LIN {X 0,Y 480.607,Z 857.054,A -85,B 0,C 180,E1 -14352.742,E2 -14352.742} C_VEL
LIN {X 0,Y 484.902,Z 835.629,A -85,B 0,C 180,E1 -14353.946,E2 -14353.946} C_VEL
LIN {X 0,Y 488.749,Z 813.876,A -85,B 0,C 180,E1 -14354.976,E2 -14354.976} C_VEL
LIN {X 0,Y 492.238,Z 790.021,A -85,B 0,C 180,E1 -14355.873,E2 -14355.873} C_VEL
LIN {X 0,Y 494.835,Z 768.166,A -85,B 0,C 180,E1 -14356.519,E2 -14356.519} C_VEL
LIN {X 0,Y 497.066,Z 742.106,A -85,B 0,C 180,E1 -14357.081,E2 -14357.081} C_VEL
LIN {X 0,Y 507.784,Z 512.286,A -85,B 0,C 180,E1 -14360.624,E2 -14360.624} C_VEL
LIN {X 0,Y 509.838,Z 466.585,A -85,B 0,C 180,E1 -14361.344,E2 -14361.344} C_VEL
LIN {X 0,Y 502.67,Z 455.07,A -85,B 0,C 180,E1 -14362.649,E2 -14362.649} C_VEL
LIN {X 0,Y 491.609,Z 438.773,A -85,B 0,C 180,E1 -14364.787,E2 -14364.787} C_VEL
LIN {X 0,Y 480.959,Z 424.124,A -85,B 0,C 180,E1 -14367.032,E2 -14367.032} C_VEL
LIN {X 0,Y 472.701,Z 413.452,A -85,B 0,C 180,E1 -14368.927,E2 -14368.927} C_VEL
LIN {X 0,Y 468.353,Z 407.951,A -85,B 0,C 180,E1 -14369.993,E2 -14369.993} C_VEL
LIN {X 0,Y 464.571,Z 403.2,A -85,B 0,C 180,E1 -14370.965,E2 -14370.965} C_VEL
LIN {X 0,Y 460.387,Z 398.04,A -85,B 0,C 180,E1 -14372.093,E2 -14372.093} C_VEL
LIN {X 0,Y 456.745,Z 393.676,A -85,B 0,C 180,E1 -14373.124,E2 -14373.124} C_VEL
LIN {X 0,Y 455.561,Z 392.247,A -85,B 0,C 180,E1 -14373.471,E2 -14373.471} C_VEL
LIN {X 0,Y 452.156,Z 388.527,A -85,B 0,C 180,E1 -14374.49,E2 -14374.49} C_VEL
LIN {X 0,Y 450.792,Z 386.471,A -85,B 0,C 180,E1 -14374.934,E2 -14374.934} C_VEL
LIN {X 0,Y 447.515,Z 383.478,A -85,B 0,C 180,E1 -14375.971,E2 -14375.971} C_VEL
LIN {X 0,Y 445.396,Z 380.169,A -85,B 0,C 180,E1 -14376.727,E2 -14376.727} C_VEL
LIN {X 0,Y 442.222,Z 377.701,A -85,B 0,C 180,E1 -14377.815,E2 -14377.815} C_VEL
LIN {X 0,Y 440.297,Z 374.242,A -85,B 0,C 180,E1 -14378.595,E2 -14378.595} C_VEL
LIN {X 0,Y 439.743,Z 373.706,A -85,B 0,C 180,E1 -14378.805,E2 -14378.805} C_VEL
LIN {X 0,Y 436.653,Z 371.721,A -85,B 0,C 180,E1 -14379.98,E2 -14379.98} C_VEL
LIN {X 0,Y 434.814,Z 368.919,A -85,B 0,C 180,E1 -14380.801,E2 -14380.801} C_VEL
LIN {X 0,Y 434.363,Z 367.099,A -85,B 0,C 180,E1 -14381.105,E2 -14381.105} C_VEL
LIN {X 0,Y 434.359,Z 367.094,A -85,B 0,C 180,E1 -14384.922,E2 -14384.922} C_VEL
LIN {X 0,Y 434.379,Z 367.091,A -85,B 0,C 180,E1 -14388.582,E2 -14388.582} C_VEL
LIN {X 0,Y 434.41,Z 367.102,A -85,B 0,C 180,E1 -14392.328,E2 -14392.328} C_VEL
LIN {X 0,Y 434.406,Z 367.121,A -85,B 0,C 180,E1 -14396.173,E2 -14396.173} C_VEL
LIN {X 0,Y 434.379,Z 367.105,A -85,B 0,C 180,E1 -14399.868,E2 -14399.868} C_VEL
LIN {X 0,Y 434.36,Z 367.091,A -85,B 0,C 180,E1 -14403.563,E2 -14403.563} C_VEL
LIN {X 0,Y 434.358,Z 367.094,A -85,B 0,C 180,E1 -14407.274,E2 -14407.274} C_VEL
LIN {X 0,Y 434.385,Z 367.106,A -85,B 0,C 180,E1 -14410.88,E2 -14410.88} C_VEL
LIN {X 0,Y 434.417,Z 367.117,A -85,B 0,C 180,E1 -14414.666,E2 -14414.666} C_VEL
LIN {X 0,Y 434.406,Z 367.116,A -85,B 0,C 180,E1 -14418.52,E2 -14418.52} C_VEL
LIN {X 0,Y 434.457,Z 367.443,A -85,B 0,C 180,E1 -14418.657,E2 -14418.657} C_VEL
LIN {X 0,Y 435.442,Z 370.22,A -85,B 0,C 180,E1 -14419.17,E2 -14419.17} C_VEL
LIN {X 0,Y 437.864,Z 372.753,A -85,B 0,C 180,E1 -14420.171,E2 -14420.171} C_VEL
LIN {X 0,Y 440.192,Z 374.091,A -85,B 0,C 180,E1 -14421.032,E2 -14421.032} C_VEL
LIN {X 0,Y 442.012,Z 377.461,A -85,B 0,C 180,E1 -14421.777,E2 -14421.777} C_VEL
LIN {X 0,Y 445.345,Z 380.151,A -85,B 0,C 180,E1 -14422.926,E2 -14422.926} C_VEL
LIN {X 0,Y 448.828,Z 384.901,A -85,B 0,C 180,E1 -14424.129,E2 -14424.129} C_VEL
LIN {X 0,Y 450.868,Z 387.155,A -85,B 0,C 180,E1 -14424.781,E2 -14424.781} C_VEL
LIN {X 0,Y 454.843,Z 392.158,A -85,B 0,C 180,E1 -14426.012,E2 -14426.012} C_VEL
LIN {X 0,Y 459.096,Z 397.573,A -85,B 0,C 180,E1 -14427.253,E2 -14427.253} C_VEL
LIN {X 0,Y 466.167,Z 406.901,A -85,B 0,C 180,E1 -14429.172,E2 -14429.172} C_VEL
LIN {X 0,Y 473.965,Z 417.836,A -85,B 0,C 180,E1 -14431.122,E2 -14431.122} C_VEL
LIN {X 0,Y 482.316,Z 429.887,A -85,B 0,C 180,E1 -14433.04,E2 -14433.04} C_VEL
LIN {X 0,Y 491.291,Z 443.78,A -85,B 0,C 180,E1 -14434.954,E2 -14434.954} C_VEL
LIN {X 0,Y 501.111,Z 459.807,A -85,B 0,C 180,E1 -14436.895,E2 -14436.895} C_VEL
LIN {X 0,Y 509.771,Z 475.225,A -85,B 0,C 180,E1 -14438.507,E2 -14438.507} C_VEL
LIN {X 0,Y 498.368,Z 722.255,A -85,B 0,C 180,E1 -14442.296,E2 -14442.296} C_VEL
LIN {X 0,Y 496.144,Z 766.257,A -85,B 0,C 180,E1 -14443.004,E2 -14443.004} C_VEL
LIN {X 0,Y 493.733,Z 790.305,A -85,B 0,C 180,E1 -14443.551,E2 -14443.551} C_VEL
LIN {X 0,Y 490.946,Z 811.995,A -85,B 0,C 180,E1 -14444.195,E2 -14444.195} C_VEL
LIN {X 0,Y 487.211,Z 835.448,A -85,B 0,C 180,E1 -14445.091,E2 -14445.091} C_VEL
LIN {X 0,Y 483.594,Z 855.156,A -85,B 0,C 180,E1 -14446.016,E2 -14446.016} C_VEL
LIN {X 0,Y 478.87,Z 878.071,A -85,B 0,C 180,E1 -14447.306,E2 -14447.306} C_VEL
LIN {X 0,Y 474.326,Z 897.652,A -85,B 0,C 180,E1 -14448.63,E2 -14448.63} C_VEL
LIN {X 0,Y 469.589,Z 916.875,A -85,B 0,C 180,E1 -14450.14,E2 -14450.14} C_VEL
LIN {X 0,Y 464.072,Z 937.548,A -85,B 0,C 180,E1 -14452.054,E2 -14452.054} C_VEL
LIN {X 0,Y 459.269,Z 954.903,A -85,B 0,C 180,E1 -14453.92,E2 -14453.92} C_VEL
LIN {X 0,Y 453.924,Z 973.715,A -85,B 0,C 180,E1 -14456.282,E2 -14456.282} C_VEL
LIN {X 0,Y 449.837,Z 988.033,A -85,B 0,C 180,E1 -14458.36,E2 -14458.36} C_VEL
LIN {X 0,Y 445.405,Z 1003.835,A -85,B 0,C 180,E1 -14460.994,E2 -14460.994} C_VEL
LIN {X 0,Y 441.88,Z 1016.82,A -85,B 0,C 180,E1 -14463.527,E2 -14463.527} C_VEL
LIN {X 0,Y 438.683,Z 1029.589,A -85,B 0,C 180,E1 -14466.389,E2 -14466.389} C_VEL
LIN {X 0,Y 436.18,Z 1040.548,A -85,B 0,C 180,E1 -14469.327,E2 -14469.327} C_VEL
LIN {X 0,Y 434.432,Z 1049.638,A -85,B 0,C 180,E1 -14472.175,E2 -14472.175} C_VEL
LIN {X 0,Y 433.099,Z 1058.109,A -85,B 0,C 180,E1 -14475.425,E2 -14475.425} C_VEL
LIN {X 0,Y 432.416,Z 1064.059,A -85,B 0,C 180,E1 -14478.259,E2 -14478.259} C_VEL
LIN {X 0,Y 432.041,Z 1069.434,A -85,B 0,C 180,E1 -14481.616,E2 -14481.616} C_VEL
LIN {X 0,Y 431.949,Z 1072.492,A -85,B 0,C 180,E1 -14484.421,E2 -14484.421} C_VEL
LIN {X 0,Y 431.945,Z 1074.289,A -85,B 0,C 180,E1 -14487.081,E2 -14487.081} C_VEL
LIN {X 0,Y 431.946,Z 1074.998,A -85,B 0,C 180,E1 -14490.265,E2 -14490.265} C_VEL
LIN {X 0,Y 431.947,Z 1074.217,A -85,B 0,C 180,E1 -14493.052,E2 -14493.052} C_VEL
LIN {X 0,Y 431.952,Z 1072.37,A -85,B 0,C 180,E1 -14495.712,E2 -14495.712} C_VEL
LIN {X 0,Y 432.06,Z 1068.893,A -85,B 0,C 180,E1 -14498.816,E2 -14498.816} C_VEL
LIN {X 0,Y 432.44,Z 1063.789,A -85,B 0,C 180,E1 -14501.875,E2 -14501.875} C_VEL
LIN {X 0,Y 433.14,Z 1057.785,A -85,B 0,C 180,E1 -14504.71,E2 -14504.71} C_VEL
LIN {X 0,Y 434.569,Z 1048.793,A -85,B 0,C 180,E1 -14508.096,E2 -14508.096} C_VEL
LIN {X 0,Y 436.279,Z 1040.061,A -85,B 0,C 180,E1 -14510.808,E2 -14510.808} C_VEL
LIN {X 0,Y 438.984,Z 1028.25,A -85,B 0,C 180,E1 -14513.918,E2 -14513.918} C_VEL
LIN {X 0,Y 442.043,Z 1016.141,A -85,B 0,C 180,E1 -14516.607,E2 -14516.607} C_VEL
LIN {X 0,Y 446.02,Z 1001.585,A -85,B 0,C 180,E1 -14519.403,E2 -14519.403} C_VEL
LIN {X 0,Y 450.069,Z 987.118,A -85,B 0,C 180,E1 -14521.771,E2 -14521.771} C_VEL
LIN {X 0,Y 454.46,Z 971.776,A -85,B 0,C 180,E1 -14523.976,E2 -14523.976} C_VEL
LIN {X 0,Y 459.719,Z 953.135,A -85,B 0,C 180,E1 -14526.271,E2 -14526.271} C_VEL
LIN {X 0,Y 464.436,Z 936.092,A -85,B 0,C 180,E1 -14528.083,E2 -14528.083} C_VEL
LIN {X 0,Y 470.052,Z 914.786,A -85,B 0,C 180,E1 -14530.022,E2 -14530.022} C_VEL
LIN {X 0,Y 474.493,Z 896.72,A -85,B 0,C 180,E1 -14531.428,E2 -14531.428} C_VEL
LIN {X 0,Y 479.379,Z 875.572,A -85,B 0,C 180,E1 -14532.841,E2 -14532.841} C_VEL
LIN {X 0,Y 483.777,Z 853.85,A -85,B 0,C 180,E1 -14534.042,E2 -14534.042} C_VEL
LIN {X 0,Y 487.42,Z 833.905,A -85,B 0,C 180,E1 -14534.967,E2 -14534.967} C_VEL
LIN {X 0,Y 491.276,Z 808.969,A -85,B 0,C 180,E1 -14535.894,E2 -14535.894} C_VEL
LIN {X 0,Y 493.87,Z 788.534,A -85,B 0,C 180,E1 -14536.486,E2 -14536.486} C_VEL
LIN {X 0,Y 496.258,Z 763.311,A -85,B 0,C 180,E1 -14537.04,E2 -14537.04} C_VEL
LIN {X 0,Y 499.532,Z 694.355,A -85,B 0,C 180,E1 -14538.123,E2 -14538.123} C_VEL
LIN {X 0,Y 509.617,Z 474.877,A -85,B 0,C 180,E1 -14541.5,E2 -14541.5} C_VEL
LIN {X 0,Y 498.824,Z 456.036,A -85,B 0,C 180,E1 -14543.517,E2 -14543.517} C_VEL
LIN {X 0,Y 487.736,Z 438.217,A -85,B 0,C 180,E1 -14545.754,E2 -14545.754} C_VEL
LIN {X 0,Y 476.706,Z 421.573,A -85,B 0,C 180,E1 -14548.197,E2 -14548.197} C_VEL
LIN {X 0,Y 467.195,Z 408.431,A -85,B 0,C 180,E1 -14550.512,E2 -14550.512} C_VEL
LIN {X 0,Y 461.589,Z 400.928,A -85,B 0,C 180,E1 -14551.997,E2 -14551.997} C_VEL
LIN {X 0,Y 457.333,Z 395.328,A -85,B 0,C 180,E1 -14553.196,E2 -14553.196} C_VEL
LIN {X 0,Y 452.168,Z 388.749,A -85,B 0,C 180,E1 -14554.746,E2 -14554.746} C_VEL
LIN {X 0,Y 449.208,Z 385.26,A -85,B 0,C 180,E1 -14555.682,E2 -14555.682} C_VEL
LIN {X 0,Y 446.351,Z 381.674,A -85,B 0,C 180,E1 -14556.64,E2 -14556.64} C_VEL
LIN {X 0,Y 445.112,Z 380.025,A -85,B 0,C 180,E1 -14557.074,E2 -14557.074} C_VEL
LIN {X 0,Y 441.822,Z 377.223,A -85,B 0,C 180,E1 -14558.213,E2 -14558.213} C_VEL
LIN {X 0,Y 440.006,Z 373.768,A -85,B 0,C 180,E1 -14558.958,E2 -14558.958} C_VEL
LIN {X 0,Y 436.552,Z 371.673,A -85,B 0,C 180,E1 -14560.255,E2 -14560.255} C_VEL
LIN {X 0,Y 434.855,Z 368.973,A -85,B 0,C 180,E1 -14561.012,E2 -14561.012} C_VEL
LIN {X 0,Y 434.41,Z 367.108,A -85,B 0,C 180,E1 -14561.306,E2 -14561.306} C_VEL
LIN {X 0,Y 434.389,Z 367.101,A -85,B 0,C 180,E1 -14565.06,E2 -14565.06} C_VEL
LIN {X 0,Y 434.365,Z 367.094,A -85,B 0,C 180,E1 -14568.716,E2 -14568.716} C_VEL
LIN {X 0,Y 434.361,Z 367.092,A -85,B 0,C 180,E1 -14572.46,E2 -14572.46} C_VEL
LIN {X 0,Y 434.378,Z 367.102,A -85,B 0,C 180,E1 -14576.172,E2 -14576.172} C_VEL
LIN {X 0,Y 434.412,Z 367.12,A -85,B 0,C 180,E1 -14579.868,E2 -14579.868} C_VEL
LIN {X 0,Y 434.407,Z 367.106,A -85,B 0,C 180,E1 -14583.695,E2 -14583.695} C_VEL
LIN {X 0,Y 434.387,Z 367.09,A -85,B 0,C 180,E1 -14587.406,E2 -14587.406} C_VEL
LIN {X 0,Y 434.365,Z 367.093,A -85,B 0,C 180,E1 -14591.015,E2 -14591.015} C_VEL
LIN {X 0,Y 434.368,Z 367.102,A -85,B 0,C 180,E1 -14594.804,E2 -14594.804} C_VEL
LIN {X 0,Y 434.386,Z 367.113,A -85,B 0,C 180,E1 -14598.521,E2 -14598.521} C_VEL
LIN {X 0,Y 434.391,Z 367.263,A -85,B 0,C 180,E1 -14599.146,E2 -14599.146} C_VEL
LIN {X 0,Y 435.315,Z 369.953,A -85,B 0,C 180,E1 -14599.629,E2 -14599.629} C_VEL
LIN {X 0,Y 437.809,Z 372.717,A -85,B 0,C 180,E1 -14600.662,E2 -14600.662} C_VEL
LIN {X 0,Y 440.238,Z 374.085,A -85,B 0,C 180,E1 -14601.554,E2 -14601.554} C_VEL
LIN {X 0,Y 442.066,Z 377.526,A -85,B 0,C 180,E1 -14602.298,E2 -14602.298} C_VEL
LIN {X 0,Y 444.961,Z 379.949,A -85,B 0,C 180,E1 -14603.297,E2 -14603.297} C_VEL
LIN {X 0,Y 445.862,Z 380.7,A -85,B 0,C 180,E1 -14603.597,E2 -14603.597} C_VEL
LIN {X 0,Y 448.273,Z 384.397,A -85,B 0,C 180,E1 -14604.442,E2 -14604.442} C_VEL
LIN {X 0,Y 451.31,Z 387.146,A -85,B 0,C 180,E1 -14605.386,E2 -14605.386} C_VEL
LIN {X 0,Y 454.326,Z 391.184,A -85,B 0,C 180,E1 -14606.325,E2 -14606.325} C_VEL
LIN {X 0,Y 456.534,Z 393.368,A -85,B 0,C 180,E1 -14606.96,E2 -14606.96} C_VEL
LIN {X 0,Y 459.957,Z 397.656,A -85,B 0,C 180,E1 -14607.935,E2 -14607.935} C_VEL
LIN {X 0,Y 461.627,Z 399.54,A -85,B 0,C 180,E1 -14608.388,E2 -14608.388} C_VEL
LIN {X 0,Y 466.733,Z 405.915,A -85,B 0,C 180,E1 -14609.732,E2 -14609.732} C_VEL
LIN {X 0,Y 471.262,Z 411.659,A -85,B 0,C 180,E1 -14610.859,E2 -14610.859} C_VEL
LIN {X 0,Y 478.641,Z 421.069,A -85,B 0,C 180,E1 -14612.578,E2 -14612.578} C_VEL
LIN {X 0,Y 489.178,Z 435.437,A -85,B 0,C 180,E1 -14614.841,E2 -14614.841} C_VEL
LIN {X 0,Y 500.544,Z 451.857,A -85,B 0,C 180,E1 -14617.069,E2 -14617.069} C_VEL
LIN {X 0,Y 509.147,Z 465.502,A -85,B 0,C 180,E1 -14618.646,E2 -14618.646} C_VEL
LIN {X 0,Y 509.876,Z 467.057,A -85,B 0,C 180,E1 -14618.784,E2 -14618.784} C_VEL
LIN {X 0,Y 498.05,Z 722.14,A -85,B 0,C 180,E1 -14622.693,E2 -14622.693} C_VEL
LIN {X 0,Y 496.16,Z 753.273,A -85,B 0,C 180,E1 -14623.235,E2 -14623.235} C_VEL
LIN {X 0,Y 494.016,Z 774.953,A -85,B 0,C 180,E1 -14623.763,E2 -14623.763} C_VEL
LIN {X 0,Y 490.73,Z 800.447,A -85,B 0,C 180,E1 -14624.592,E2 -14624.592} C_VEL
LIN {X 0,Y 487.43,Z 821.156,A -85,B 0,C 180,E1 -14625.448,E2 -14625.448} C_VEL
LIN {X 0,Y 483.211,Z 844.209,A -85,B 0,C 180,E1 -14626.607,E2 -14626.607} C_VEL
LIN {X 0,Y 478.889,Z 864.397,A -85,B 0,C 180,E1 -14627.836,E2 -14627.836} C_VEL
LIN {X 0,Y 474.078,Z 885.286,A -85,B 0,C 180,E1 -14629.329,E2 -14629.329} C_VEL
LIN {X 0,Y 468.947,Z 905.227,A -85,B 0,C 180,E1 -14631.024,E2 -14631.024} C_VEL
LIN {X 0,Y 464.194,Z 922.816,A -85,B 0,C 180,E1 -14632.751,E2 -14632.751} C_VEL
LIN {X 0,Y 458.768,Z 941.82,A -85,B 0,C 180,E1 -14634.93,E2 -14634.93} C_VEL
LIN {X 0,Y 454.185,Z 957.46,A -85,B 0,C 180,E1 -14637.011,E2 -14637.011} C_VEL
LIN {X 0,Y 449.179,Z 974.473,A -85,B 0,C 180,E1 -14639.648,E2 -14639.648} C_VEL
LIN {X 0,Y 445.35,Z 987.585,A -85,B 0,C 180,E1 -14642.015,E2 -14642.015} C_VEL
LIN {X 0,Y 441.421,Z 1001.642,A -85,B 0,C 180,E1 -14644.968,E2 -14644.968} C_VEL
LIN {X 0,Y 438.583,Z 1012.347,A -85,B 0,C 180,E1 -14647.621,E2 -14647.621} C_VEL
LIN {X 0,Y 436.08,Z 1023.008,A -85,B 0,C 180,E1 -14650.721,E2 -14650.721} C_VEL
LIN {X 0,Y 434.355,Z 1031.358,A -85,B 0,C 180,E1 -14653.689,E2 -14653.689} C_VEL
LIN {X 0,Y 433.163,Z 1038.583,A -85,B 0,C 180,E1 -14656.79,E2 -14656.79} C_VEL
LIN {X 0,Y 432.436,Z 1044.258,A -85,B 0,C 180,E1 -14660.014,E2 -14660.014} C_VEL
LIN {X 0,Y 432.129,Z 1047.959,A -85,B 0,C 180,E1 -14662.822,E2 -14662.822} C_VEL
LIN {X 0,Y 432.054,Z 1049.16,A -85,B 0,C 180,E1 -14664.016,E2 -14664.016} C_VEL
LIN {X 0,Y 431.001,Z 1050.055,A -85,B 0,C 180,E1 -14665.031,E2 -14665.031} C_VEL
LIN {X 0,Y 426.312,Z 1051.369,A -85,B 0,C 180,E1 -14666.947,E2 -14666.947} C_VEL
LIN {X 0,Y 424.146,Z 1051.897,A -85,B 0,C 180,E1 -14668.194,E2 -14668.194} C_VEL
LIN {X 0,Y 423.955,Z 1051.968,A -85,B 0,C 180,E1 -14668.646,E2 -14668.646} C_VEL
LIN {X 0,Y 423.958,Z 1051.984,A -85,B 0,C 180,E1 -14671.352,E2 -14671.352} C_VEL
LIN {X 0,Y 424.005,Z 1050.767,A -85,B 0,C 180,E1 -14674.463,E2 -14674.463} C_VEL
LIN {X 0,Y 424.156,Z 1047.974,A -85,B 0,C 180,E1 -14677.586,E2 -14677.586} C_VEL
LIN {X 0,Y 424.506,Z 1044.214,A -85,B 0,C 180,E1 -14680.45,E2 -14680.45} C_VEL
LIN {X 0,Y 425.318,Z 1038.416,A -85,B 0,C 180,E1 -14683.736,E2 -14683.736} C_VEL
LIN {X 0,Y 426.557,Z 1031.476,A -85,B 0,C 180,E1 -14686.758,E2 -14686.758} C_VEL
LIN {X 0,Y 428.508,Z 1022.705,A -85,B 0,C 180,E1 -14689.918,E2 -14689.918} C_VEL
LIN {X 0,Y 431.068,Z 1012.367,A -85,B 0,C 180,E1 -14692.946,E2 -14692.946} C_VEL
LIN {X 0,Y 434.273,Z 1000.957,A -85,B 0,C 180,E1 -14695.808,E2 -14695.808} C_VEL
LIN {X 0,Y 438.198,Z 987.585,A -85,B 0,C 180,E1 -14698.632,E2 -14698.632} C_VEL
LIN {X 0,Y 442.219,Z 974.448,A -85,B 0,C 180,E1 -14701.033,E2 -14701.033} C_VEL
LIN {X 0,Y 447.368,Z 957.672,A -85,B 0,C 180,E1 -14703.662,E2 -14703.662} C_VEL
LIN {X 0,Y 452.053,Z 942.317,A -85,B 0,C 180,E1 -14705.731,E2 -14705.731} C_VEL
LIN {X 0,Y 457.887,Z 922.629,A -85,B 0,C 180,E1 -14708.011,E2 -14708.011} C_VEL
LIN {X 0,Y 462.685,Z 905.512,A -85,B 0,C 180,E1 -14709.705,E2 -14709.705} C_VEL
LIN {X 0,Y 468.004,Z 885.543,A -85,B 0,C 180,E1 -14711.417,E2 -14711.417} C_VEL
LIN {X 0,Y 472.925,Z 864.871,A -85,B 0,C 180,E1 -14712.906,E2 -14712.906} C_VEL
LIN {X 0,Y 477.606,Z 843.711,A -85,B 0,C 180,E1 -14714.199,E2 -14714.199} C_VEL
LIN {X 0,Y 481.741,Z 821.735,A -85,B 0,C 180,E1 -14715.307,E2 -14715.307} C_VEL
LIN {X 0,Y 485.173,Z 800.872,A -85,B 0,C 180,E1 -14716.175,E2 -14716.175} C_VEL
LIN {X 0,Y 488.609,Z 774.994,A -85,B 0,C 180,E1 -14717.02,E2 -14717.02} C_VEL
LIN {X 0,Y 490.823,Z 753.157,A -85,B 0,C 180,E1 -14717.553,E2 -14717.553} C_VEL
LIN {X 0,Y 492.819,Z 720.765,A -85,B 0,C 180,E1 -14718.115,E2 -14718.115} C_VEL
LIN {X 0,Y 504.833,Z 470.537,A -85,B 0,C 180,E1 -14721.974,E2 -14721.974} C_VEL
LIN {X 0,Y 494.554,Z 454.342,A -85,B 0,C 180,E1 -14723.924,E2 -14723.924} C_VEL
LIN {X 0,Y 483.467,Z 438.399,A -85,B 0,C 180,E1 -14726.197,E2 -14726.197} C_VEL
LIN {X 0,Y 473.671,Z 425.178,A -85,B 0,C 180,E1 -14728.396,E2 -14728.396} C_VEL
LIN {X 0,Y 465.75,Z 414.967,A -85,B 0,C 180,E1 -14730.34,E2 -14730.34} C_VEL
LIN {X 0,Y 461.801,Z 410.002,A -85,B 0,C 180,E1 -14731.376,E2 -14731.376} C_VEL
LIN {X 0,Y 457.778,Z 405.021,A -85,B 0,C 180,E1 -14732.486,E2 -14732.486} C_VEL
LIN {X 0,Y 454.017,Z 400.251,A -85,B 0,C 180,E1 -14733.585,E2 -14733.585} C_VEL
LIN {X 0,Y 449.874,Z 395.681,A -85,B 0,C 180,E1 -14734.845,E2 -14734.845} C_VEL
LIN {X 0,Y 448.515,Z 393.78,A -85,B 0,C 180,E1 -14735.291,E2 -14735.291} C_VEL
LIN {X 0,Y 445.049,Z 390.259,A -85,B 0,C 180,E1 -14736.427,E2 -14736.427} C_VEL
LIN {X 0,Y 443.377,Z 387.689,A -85,B 0,C 180,E1 -14737.036,E2 -14737.036} C_VEL
LIN {X 0,Y 440.106,Z 384.859,A -85,B 0,C 180,E1 -14738.194,E2 -14738.194} C_VEL
LIN {X 0,Y 438.141,Z 381.457,A -85,B 0,C 180,E1 -14739.004,E2 -14739.004} C_VEL
LIN {X 0,Y 434.79,Z 379.107,A -85,B 0,C 180,E1 -14740.311,E2 -14740.311} C_VEL
LIN {X 0,Y 432.787,Z 375.962,A -85,B 0,C 180,E1 -14741.233,E2 -14741.233} C_VEL
LIN {X 0,Y 432.209,Z 374.803,A -85,B 0,C 180,E1 -14741.522,E2 -14741.522} C_VEL
LIN {X 0,Y 428.816,Z 372.879,A -85,B 0,C 180,E1 -14743.054,E2 -14743.054} C_VEL
LIN {X 0,Y 426.978,Z 370.049,A -85,B 0,C 180,E1 -14744.063,E2 -14744.063} C_VEL
LIN {X 0,Y 426.441,Z 368.079,A -85,B 0,C 180,E1 -14744.496,E2 -14744.496} C_VEL
LIN {X 0,Y 426.465,Z 368.081,A -85,B 0,C 180,E1 -14748.23,E2 -14748.23} C_VEL
LIN {X 0,Y 426.481,Z 368.092,A -85,B 0,C 180,E1 -14752.185,E2 -14752.185} C_VEL
LIN {X 0,Y 426.464,Z 368.111,A -85,B 0,C 180,E1 -14756.101,E2 -14756.101} C_VEL
LIN {X 0,Y 426.44,Z 368.092,A -85,B 0,C 180,E1 -14759.866,E2 -14759.866} C_VEL
LIN {X 0,Y 426.423,Z 368.08,A -85,B 0,C 180,E1 -14763.63,E2 -14763.63} C_VEL
LIN {X 0,Y 426.418,Z 368.081,A -85,B 0,C 180,E1 -14767.41,E2 -14767.41} C_VEL
LIN {X 0,Y 426.426,Z 368.09,A -85,B 0,C 180,E1 -14771.223,E2 -14771.223} C_VEL
LIN {X 0,Y 426.447,Z 368.1,A -85,B 0,C 180,E1 -14774.979,E2 -14774.979} C_VEL
LIN {X 0,Y 426.456,Z 368.293,A -85,B 0,C 180,E1 -14775.247,E2 -14775.247} C_VEL
LIN {X 0,Y 427.321,Z 370.893,A -85,B 0,C 180,E1 -14775.819,E2 -14775.819} C_VEL
LIN {X 0,Y 429.991,Z 373.788,A -85,B 0,C 180,E1 -14777.177,E2 -14777.177} C_VEL
LIN {X 0,Y 432.52,Z 375.161,A -85,B 0,C 180,E1 -14778.29,E2 -14778.29} C_VEL
LIN {X 0,Y 434.16,Z 378.422,A -85,B 0,C 180,E1 -14779.089,E2 -14779.089} C_VEL
LIN {X 0,Y 436.932,Z 380.842,A -85,B 0,C 180,E1 -14780.216,E2 -14780.216} C_VEL
LIN {X 0,Y 438.24,Z 381.718,A -85,B 0,C 180,E1 -14780.711,E2 -14780.711} C_VEL
LIN {X 0,Y 440.548,Z 385.401,A -85,B 0,C 180,E1 -14781.643,E2 -14781.643} C_VEL
LIN {X 0,Y 443.841,Z 388.254,A -85,B 0,C 180,E1 -14782.798,E2 -14782.798} C_VEL
LIN {X 0,Y 446.775,Z 392.266,A -85,B 0,C 180,E1 -14783.826,E2 -14783.826} C_VEL
LIN {X 0,Y 449.151,Z 395.008,A -85,B 0,C 180,E1 -14784.601,E2 -14784.601} C_VEL
LIN {X 0,Y 452.706,Z 399.589,A -85,B 0,C 180,E1 -14785.722,E2 -14785.722} C_VEL
LIN {X 0,Y 456.806,Z 404.898,A -85,B 0,C 180,E1 -14786.943,E2 -14786.943} C_VEL
LIN {X 0,Y 463.479,Z 413.79,A -85,B 0,C 180,E1 -14788.792,E2 -14788.792} C_VEL
LIN {X 0,Y 471.505,Z 425.231,A -85,B 0,C 180,E1 -14790.842,E2 -14790.842} C_VEL
LIN {X 0,Y 479.65,Z 437.222,A -85,B 0,C 180,E1 -14792.749,E2 -14792.749} C_VEL
LIN {X 0,Y 487.804,Z 449.977,A -85,B 0,C 180,E1 -14794.525,E2 -14794.525} C_VEL
LIN {X 0,Y 497.797,Z 466.497,A -85,B 0,C 180,E1 -14796.546,E2 -14796.546} C_VEL
LIN {X 0,Y 504.611,Z 478.946,A -85,B 0,C 180,E1 -14797.854,E2 -14797.854} C_VEL
LIN {X 0,Y 492.829,Z 725.76,A -85,B 0,C 180,E1 -14801.663,E2 -14801.663} C_VEL
LIN {X 0,Y 490.655,Z 766.549,A -85,B 0,C 180,E1 -14802.328,E2 -14802.328} C_VEL
LIN {X 0,Y 488.213,Z 790.233,A -85,B 0,C 180,E1 -14802.871,E2 -14802.871} C_VEL
LIN {X 0,Y 485.285,Z 812.344,A -85,B 0,C 180,E1 -14803.53,E2 -14803.53} C_VEL
LIN {X 0,Y 481.518,Z 835.24,A -85,B 0,C 180,E1 -14804.412,E2 -14804.412} C_VEL
LIN {X 0,Y 477.845,Z 854.651,A -85,B 0,C 180,E1 -14805.325,E2 -14805.325} C_VEL
LIN {X 0,Y 473.031,Z 877.404,A -85,B 0,C 180,E1 -14806.608,E2 -14806.608} C_VEL
LIN {X 0,Y 468.194,Z 897.557,A -85,B 0,C 180,E1 -14807.978,E2 -14807.978} C_VEL
LIN {X 0,Y 463.14,Z 917.4,A -85,B 0,C 180,E1 -14809.552,E2 -14809.552} C_VEL
LIN {X 0,Y 457.651,Z 937.208,A -85,B 0,C 180,E1 -14811.408,E2 -14811.408} C_VEL
LIN {X 0,Y 452.789,Z 954.127,A -85,B 0,C 180,E1 -14813.241,E2 -14813.241} C_VEL
LIN {X 0,Y 447.059,Z 973.497,A -85,B 0,C 180,E1 -14815.693,E2 -14815.693} C_VEL
LIN {X 0,Y 442.595,Z 988.519,A -85,B 0,C 180,E1 -14817.907,E2 -14817.907} C_VEL
LIN {X 0,Y 437.688,Z 1005.214,A -85,B 0,C 180,E1 -14820.771,E2 -14820.771} C_VEL
LIN {X 0,Y 434.12,Z 1017.887,A -85,B 0,C 180,E1 -14823.312,E2 -14823.312} C_VEL
LIN {X 0,Y 430.505,Z 1031.68,A -85,B 0,C 180,E1 -14826.554,E2 -14826.554} C_VEL
LIN {X 0,Y 428.153,Z 1041.727,A -85,B 0,C 180,E1 -14829.351,E2 -14829.351} C_VEL
LIN {X 0,Y 426.143,Z 1051.913,A -85,B 0,C 180,E1 -14832.742,E2 -14832.742} C_VEL
LIN {X 0,Y 425.055,Z 1058.818,A -85,B 0,C 180,E1 -14835.561,E2 -14835.561} C_VEL
LIN {X 0,Y 424.342,Z 1065.138,A -85,B 0,C 180,E1 -14838.722,E2 -14838.722} C_VEL
LIN {X 0,Y 424.017,Z 1069.708,A -85,B 0,C 180,E1 -14841.866,E2 -14841.866} C_VEL
LIN {X 0,Y 423.949,Z 1072.51,A -85,B 0,C 180,E1 -14844.587,E2 -14844.587} C_VEL
LIN {X 0,Y 423.946,Z 1074.421,A -85,B 0,C 180,E1 -14847.702,E2 -14847.702} C_VEL
LIN {X 0,Y 423.949,Z 1074.693,A -85,B 0,C 180,E1 -14850.811,E2 -14850.811} C_VEL
LIN {X 0,Y 423.943,Z 1073.794,A -85,B 0,C 180,E1 -14853.516,E2 -14853.516} C_VEL
LIN {X 0,Y 423.957,Z 1071.573,A -85,B 0,C 180,E1 -14856.5,E2 -14856.5} C_VEL
LIN {X 0,Y 424.151,Z 1067.418,A -85,B 0,C 180,E1 -14859.805,E2 -14859.805} C_VEL
LIN {X 0,Y 424.59,Z 1062.534,A -85,B 0,C 180,E1 -14862.651,E2 -14862.651} C_VEL
LIN {X 0,Y 425.574,Z 1055.284,A -85,B 0,C 180,E1 -14865.955,E2 -14865.955} C_VEL
LIN {X 0,Y 427.01,Z 1047.163,A -85,B 0,C 180,E1 -14868.913,E2 -14868.913} C_VEL
LIN {X 0,Y 429.229,Z 1037.034,A -85,B 0,C 180,E1 -14872.027,E2 -14872.027} C_VEL
LIN {X 0,Y 432.167,Z 1025.121,A -85,B 0,C 180,E1 -14875.049,E2 -14875.049} C_VEL
LIN {X 0,Y 435.825,Z 1011.821,A -85,B 0,C 180,E1 -14877.958,E2 -14877.958} C_VEL
LIN {X 0,Y 439.917,Z 997.465,A -85,B 0,C 180,E1 -14880.606,E2 -14880.606} C_VEL
LIN {X 0,Y 444.324,Z 982.624,A -85,B 0,C 180,E1 -14882.996,E2 -14882.996} C_VEL
LIN {X 0,Y 449.491,Z 965.219,A -85,B 0,C 180,E1 -14885.394,E2 -14885.394} C_VEL
LIN {X 0,Y 454.249,Z 948.994,A -85,B 0,C 180,E1 -14887.332,E2 -14887.332} C_VEL
LIN {X 0,Y 460.122,Z 928.152,A -85,B 0,C 180,E1 -14889.467,E2 -14889.467} C_VEL
LIN {X 0,Y 465.015,Z 909.858,A -85,B 0,C 180,E1 -14891.063,E2 -14891.063} C_VEL
LIN {X 0,Y 470.442,Z 888.084,A -85,B 0,C 180,E1 -14892.688,E2 -14892.688} C_VEL
LIN {X 0,Y 475.069,Z 867.65,A -85,B 0,C 180,E1 -14893.96,E2 -14893.96} C_VEL
LIN {X 0,Y 479.635,Z 845.284,A -85,B 0,C 180,E1 -14895.137,E2 -14895.137} C_VEL
LIN {X 0,Y 483.594,Z 822.338,A -85,B 0,C 180,E1 -14896.101,E2 -14896.101} C_VEL
LIN {X 0,Y 487.143,Z 798.485,A -85,B 0,C 180,E1 -14896.903,E2 -14896.903} C_VEL
LIN {X 0,Y 489.853,Z 774.082,A -85,B 0,C 180,E1 -14897.505,E2 -14897.505} C_VEL
LIN {X 0,Y 491.668,Z 749.438,A -85,B 0,C 180,E1 -14897.962,E2 -14897.962} C_VEL
LIN {X 0,Y 503.52,Z 499.125,A -85,B 0,C 180,E1 -14901.825,E2 -14901.825} C_VEL
LIN {X 0,Y 504.44,Z 478.503,A -85,B 0,C 180,E1 -14902.158,E2 -14902.158} C_VEL
LIN {X 0,Y 494.16,Z 460.455,A -85,B 0,C 180,E1 -14904.142,E2 -14904.142} C_VEL
LIN {X 0,Y 483.807,Z 443.704,A -85,B 0,C 180,E1 -14906.295,E2 -14906.295} C_VEL
LIN {X 0,Y 473.646,Z 428.16,A -85,B 0,C 180,E1 -14908.607,E2 -14908.607} C_VEL
LIN {X 0,Y 463.959,Z 414.557,A -85,B 0,C 180,E1 -14911.029,E2 -14911.029} C_VEL
LIN {X 0,Y 458.961,Z 407.824,A -85,B 0,C 180,E1 -14912.387,E2 -14912.387} C_VEL
LIN {X 0,Y 454.669,Z 402.14,A -85,B 0,C 180,E1 -14913.626,E2 -14913.626} C_VEL
LIN {X 0,Y 449.718,Z 395.716,A -85,B 0,C 180,E1 -14915.152,E2 -14915.152} C_VEL
LIN {X 0,Y 446.775,Z 392.277,A -85,B 0,C 180,E1 -14916.104,E2 -14916.104} C_VEL
LIN {X 0,Y 443.827,Z 388.249,A -85,B 0,C 180,E1 -14917.131,E2 -14917.131} C_VEL
LIN {X 0,Y 439.627,Z 384.257,A -85,B 0,C 180,E1 -14918.625,E2 -14918.625} C_VEL
LIN {X 0,Y 438.052,Z 381.387,A -85,B 0,C 180,E1 -14919.28,E2 -14919.28} C_VEL
LIN {X 0,Y 434.683,Z 379.054,A -85,B 0,C 180,E1 -14920.586,E2 -14920.586} C_VEL
LIN {X 0,Y 432.754,Z 375.864,A -85,B 0,C 180,E1 -14921.476,E2 -14921.476} C_VEL
LIN {X 0,Y 432.391,Z 374.863,A -85,B 0,C 180,E1 -14921.67,E2 -14921.67} C_VEL
LIN {X 0,Y 429.083,Z 373.077,A -85,B 0,C 180,E1 -14923.135,E2 -14923.135} C_VEL
LIN {X 0,Y 426.976,Z 370.168,A -85,B 0,C 180,E1 -14924.254,E2 -14924.254} C_VEL
LIN {X 0,Y 426.427,Z 368.087,A -85,B 0,C 180,E1 -14924.682,E2 -14924.682} C_VEL
LIN {X 0,Y 426.424,Z 368.081,A -85,B 0,C 180,E1 -14928.503,E2 -14928.503} C_VEL
LIN {X 0,Y 426.425,Z 368.08,A -85,B 0,C 180,E1 -14932.319,E2 -14932.319} C_VEL
LIN {X 0,Y 426.453,Z 368.093,A -85,B 0,C 180,E1 -14935.966,E2 -14935.966} C_VEL
LIN {X 0,Y 426.488,Z 368.108,A -85,B 0,C 180,E1 -14939.731,E2 -14939.731} C_VEL
LIN {X 0,Y 426.465,Z 368.092,A -85,B 0,C 180,E1 -14943.63,E2 -14943.63} C_VEL
LIN {X 0,Y 426.448,Z 368.078,A -85,B 0,C 180,E1 -14947.409,E2 -14947.409} C_VEL
LIN {X 0,Y 426.427,Z 368.08,A -85,B 0,C 180,E1 -14951.086,E2 -14951.086} C_VEL
LIN {X 0,Y 426.429,Z 368.09,A -85,B 0,C 180,E1 -14954.808,E2 -14954.808} C_VEL
LIN {X 0,Y 426.498,Z 368.277,A -85,B 0,C 180,E1 -14955.825,E2 -14955.825} C_VEL
LIN {X 0,Y 427.452,Z 371.084,A -85,B 0,C 180,E1 -14956.442,E2 -14956.442} C_VEL
LIN {X 0,Y 429.756,Z 373.634,A -85,B 0,C 180,E1 -14957.606,E2 -14957.606} C_VEL
LIN {X 0,Y 432.448,Z 375.035,A -85,B 0,C 180,E1 -14958.782,E2 -14958.782} C_VEL
LIN {X 0,Y 434.104,Z 378.275,A -85,B 0,C 180,E1 -14959.581,E2 -14959.581} C_VEL
LIN {X 0,Y 437.042,Z 380.926,A -85,B 0,C 180,E1 -14960.77,E2 -14960.77} C_VEL
LIN {X 0,Y 438.28,Z 381.734,A -85,B 0,C 180,E1 -14961.234,E2 -14961.234} C_VEL
LIN {X 0,Y 440.518,Z 385.382,A -85,B 0,C 180,E1 -14962.135,E2 -14962.135} C_VEL
LIN {X 0,Y 443.828,Z 388.252,A -85,B 0,C 180,E1 -14963.29,E2 -14963.29} C_VEL
LIN {X 0,Y 446.589,Z 392.143,A -85,B 0,C 180,E1 -14964.258,E2 -14964.258} C_VEL
LIN {X 0,Y 449.207,Z 394.654,A -85,B 0,C 180,E1 -14965.09,E2 -14965.09} C_VEL
LIN {X 0,Y 452.596,Z 398.921,A -85,B 0,C 180,E1 -14966.151,E2 -14966.151} C_VEL
LIN {X 0,Y 454.275,Z 400.713,A -85,B 0,C 180,E1 -14966.646,E2 -14966.646} C_VEL
LIN {X 0,Y 458.188,Z 405.401,A -85,B 0,C 180,E1 -14967.77,E2 -14967.77} C_VEL
LIN {X 0,Y 464.571,Z 413.519,A -85,B 0,C 180,E1 -14969.494,E2 -14969.494} C_VEL
LIN {X 0,Y 471.886,Z 422.797,A -85,B 0,C 180,E1 -14971.31,E2 -14971.31} C_VEL
LIN {X 0,Y 482.924,Z 437.658,A -85,B 0,C 180,E1 -14973.81,E2 -14973.81} C_VEL
LIN {X 0,Y 493.863,Z 453.488,A -85,B 0,C 180,E1 -14976.062,E2 -14976.062} C_VEL
LIN {X 0,Y 504.337,Z 469.76,A -85,B 0,C 180,E1 -14978.049,E2 -14978.049} C_VEL
LIN {X 0,Y 504.716,Z 470.989,A -85,B 0,C 180,E1 -14978.133,E2 -14978.133} C_VEL
LIN {X 0,Y 492.497,Z 725.924,A -85,B 0,C 180,E1 -14982.063,E2 -14982.063} C_VEL
LIN {X 0,Y 490.664,Z 754.032,A -85,B 0,C 180,E1 -14982.565,E2 -14982.565} C_VEL
LIN {X 0,Y 488.441,Z 775.794,A -85,B 0,C 180,E1 -14983.101,E2 -14983.101} C_VEL
LIN {X 0,Y 485.122,Z 800.672,A -85,B 0,C 180,E1 -14983.916,E2 -14983.916} C_VEL
LIN {X 0,Y 481.726,Z 821.38,A -85,B 0,C 180,E1 -14984.776,E2 -14984.776} C_VEL
LIN {X 0,Y 477.378,Z 844.432,A -85,B 0,C 180,E1 -14985.942,E2 -14985.942} C_VEL
LIN {X 0,Y 472.815,Z 865.081,A -85,B 0,C 180,E1 -14987.208,E2 -14987.208} C_VEL
LIN {X 0,Y 467.74,Z 886.374,A -85,B 0,C 180,E1 -14988.748,E2 -14988.748} C_VEL
LIN {X 0,Y 462.489,Z 906.021,A -85,B 0,C 180,E1 -14990.443,E2 -14990.443} C_VEL
LIN {X 0,Y 457.391,Z 924.245,A -85,B 0,C 180,E1 -14992.259,E2 -14992.259} C_VEL
LIN {X 0,Y 451.901,Z 942.675,A -85,B 0,C 180,E1 -14994.414,E2 -14994.414} C_VEL
LIN {X 0,Y 447.163,Z 958.236,A -85,B 0,C 180,E1 -14996.518,E2 -14996.518} C_VEL
LIN {X 0,Y 442.111,Z 974.695,A -85,B 0,C 180,E1 -14999.11,E2 -14999.11} C_VEL
LIN {X 0,Y 438.108,Z 987.807,A -85,B 0,C 180,E1 -15001.511,E2 -15001.511} C_VEL
LIN {X 0,Y 434.02,Z 1001.75,A -85,B 0,C 180,E1 -15004.481,E2 -15004.481} C_VEL
LIN {X 0,Y 431.002,Z 1012.568,A -85,B 0,C 180,E1 -15007.206,E2 -15007.206} C_VEL
LIN {X 0,Y 428.359,Z 1023.228,A -85,B 0,C 180,E1 -15010.359,E2 -15010.359} C_VEL
LIN {X 0,Y 426.527,Z 1031.577,A -85,B 0,C 180,E1 -15013.382,E2 -15013.382} C_VEL
LIN {X 0,Y 425.256,Z 1038.801,A -85,B 0,C 180,E1 -15016.54,E2 -15016.54} C_VEL
LIN {X 0,Y 424.493,Z 1044.272,A -85,B 0,C 180,E1 -15019.688,E2 -15019.688} C_VEL
LIN {X 0,Y 424.164,Z 1047.862,A -85,B 0,C 180,E1 -15022.414,E2 -15022.414} C_VEL
LIN {X 0,Y 424.006,Z 1050.71,A -85,B 0,C 180,E1 -15025.537,E2 -15025.537} C_VEL
LIN {X 0,Y 423.955,Z 1051.968,A -85,B 0,C 180,E1 -15028.646,E2 -15028.646} C_VEL
LIN {X 0,Y 422.979,Z 1052.18,A -85,B 0,C 180,E1 -15029.687,E2 -15029.687} C_VEL
LIN {X 0,Y 416.503,Z 1051.897,A -85,B 0,C 180,E1 -15032.619,E2 -15032.619} C_VEL
LIN {X 0,Y 415.978,Z 1051.54,A -85,B 0,C 180,E1 -15033.384,E2 -15033.384} C_VEL
LIN {X 0,Y 416.075,Z 1049.674,A -85,B 0,C 180,E1 -15036.208,E2 -15036.208} C_VEL
LIN {X 0,Y 416.395,Z 1045.846,A -85,B 0,C 180,E1 -15039.677,E2 -15039.677} C_VEL
LIN {X 0,Y 416.991,Z 1041.217,A -85,B 0,C 180,E1 -15042.604,E2 -15042.604} C_VEL
LIN {X 0,Y 418.066,Z 1035.063,A -85,B 0,C 180,E1 -15045.68,E2 -15045.68} C_VEL
LIN {X 0,Y 419.901,Z 1026.512,A -85,B 0,C 180,E1 -15049.04,E2 -15049.04} C_VEL
LIN {X 0,Y 422.187,Z 1017.513,A -85,B 0,C 180,E1 -15051.975,E2 -15051.975} C_VEL
LIN {X 0,Y 425.567,Z 1005.497,A -85,B 0,C 180,E1 -15055.233,E2 -15055.233} C_VEL
LIN {X 0,Y 429.135,Z 993.794,A -85,B 0,C 180,E1 -15057.926,E2 -15057.926} C_VEL
LIN {X 0,Y 433.724,Z 979.237,A -85,B 0,C 180,E1 -15060.783,E2 -15060.783} C_VEL
LIN {X 0,Y 438.336,Z 964.886,A -85,B 0,C 180,E1 -15063.193,E2 -15063.193} C_VEL
LIN {X 0,Y 444.159,Z 946.571,A -85,B 0,C 180,E1 -15065.825,E2 -15065.825} C_VEL
LIN {X 0,Y 449.076,Z 930.716,A -85,B 0,C 180,E1 -15067.774,E2 -15067.774} C_VEL
LIN {X 0,Y 455.105,Z 910.515,A -85,B 0,C 180,E1 -15069.907,E2 -15069.907} C_VEL
LIN {X 0,Y 460.085,Z 892.585,A -85,B 0,C 180,E1 -15071.518,E2 -15071.518} C_VEL
LIN {X 0,Y 465.527,Z 871.616,A -85,B 0,C 180,E1 -15073.14,E2 -15073.14} C_VEL
LIN {X 0,Y 470.222,Z 851.271,A -85,B 0,C 180,E1 -15074.45,E2 -15074.45} C_VEL
LIN {X 0,Y 474.319,Z 831.654,A -85,B 0,C 180,E1 -15075.527,E2 -15075.527} C_VEL
LIN {X 0,Y 478.545,Z 808.077,A -85,B 0,C 180,E1 -15076.593,E2 -15076.593} C_VEL
LIN {X 0,Y 481.578,Z 787.8,A -85,B 0,C 180,E1 -15077.33,E2 -15077.33} C_VEL
LIN {X 0,Y 484.525,Z 763.703,A -85,B 0,C 180,E1 -15078.02,E2 -15078.02} C_VEL
LIN {X 0,Y 486.47,Z 739.921,A -85,B 0,C 180,E1 -15078.507,E2 -15078.507} C_VEL
LIN {X 0,Y 498.501,Z 498.621,A -85,B 0,C 180,E1 -15082.265,E2 -15082.265} C_VEL
LIN {X 0,Y 499.672,Z 474.113,A -85,B 0,C 180,E1 -15082.659,E2 -15082.659} C_VEL
LIN {X 0,Y 487.767,Z 455.647,A -85,B 0,C 180,E1 -15085.007,E2 -15085.007} C_VEL
LIN {X 0,Y 475.479,Z 438.171,A -85,B 0,C 180,E1 -15087.679,E2 -15087.679} C_VEL
LIN {X 0,Y 466.63,Z 426.52,A -85,B 0,C 180,E1 -15089.8,E2 -15089.8} C_VEL
LIN {X 0,Y 459.582,Z 417.375,A -85,B 0,C 180,E1 -15091.651,E2 -15091.651} C_VEL
LIN {X 0,Y 455.194,Z 411.977,A -85,B 0,C 180,E1 -15092.883,E2 -15092.883} C_VEL
LIN {X 0,Y 450.706,Z 406.485,A -85,B 0,C 180,E1 -15094.226,E2 -15094.226} C_VEL
LIN {X 0,Y 447.079,Z 402.001,A -85,B 0,C 180,E1 -15095.383,E2 -15095.383} C_VEL
LIN {X 0,Y 442.614,Z 397.024,A -85,B 0,C 180,E1 -15096.889,E2 -15096.889} C_VEL
LIN {X 0,Y 441.375,Z 395.172,A -85,B 0,C 180,E1 -15097.349,E2 -15097.349} C_VEL
LIN {X 0,Y 438.01,Z 392.011,A -85,B 0,C 180,E1 -15098.577,E2 -15098.577} C_VEL
LIN {X 0,Y 436.212,Z 389.04,A -85,B 0,C 180,E1 -15099.329,E2 -15099.329} C_VEL
LIN {X 0,Y 432.797,Z 386.32,A -85,B 0,C 180,E1 -15100.708,E2 -15100.708} C_VEL
LIN {X 0,Y 430.665,Z 382.691,A -85,B 0,C 180,E1 -15101.734,E2 -15101.734} C_VEL
LIN {X 0,Y 427.086,Z 380.306,A -85,B 0,C 180,E1 -15103.404,E2 -15103.404} C_VEL
LIN {X 0,Y 425.194,Z 377.195,A -85,B 0,C 180,E1 -15104.485,E2 -15104.485} C_VEL
LIN {X 0,Y 424.631,Z 375.878,A -85,B 0,C 180,E1 -15104.848,E2 -15104.848} C_VEL
LIN {X 0,Y 421.002,Z 373.996,A -85,B 0,C 180,E1 -15106.96,E2 -15106.96} C_VEL
LIN {X 0,Y 419.038,Z 371.092,A -85,B 0,C 180,E1 -15108.437,E2 -15108.437} C_VEL
LIN {X 0,Y 418.482,Z 369.068,A -85,B 0,C 180,E1 -15109.057,E2 -15109.057} C_VEL
LIN {X 0,Y 418.489,Z 369.073,A -85,B 0,C 180,E1 -15112.863,E2 -15112.863} C_VEL
LIN {X 0,Y 418.513,Z 369.091,A -85,B 0,C 180,E1 -15116.576,E2 -15116.576} C_VEL
LIN {X 0,Y 418.538,Z 369.09,A -85,B 0,C 180,E1 -15120.411,E2 -15120.411} C_VEL
LIN {X 0,Y 418.526,Z 369.073,A -85,B 0,C 180,E1 -15124.385,E2 -15124.385} C_VEL
LIN {X 0,Y 418.52,Z 369.065,A -85,B 0,C 180,E1 -15128.242,E2 -15128.242} C_VEL
LIN {X 0,Y 418.55,Z 369.318,A -85,B 0,C 180,E1 -15130.739,E2 -15130.739} C_VEL
LIN {X 0,Y 419.328,Z 371.786,A -85,B 0,C 180,E1 -15131.485,E2 -15131.485} C_VEL
LIN {X 0,Y 422.13,Z 374.843,A -85,B 0,C 180,E1 -15133.423,E2 -15133.423} C_VEL
LIN {X 0,Y 424.766,Z 376.089,A -85,B 0,C 180,E1 -15134.902,E2 -15134.902} C_VEL
LIN {X 0,Y 426.205,Z 379.176,A -85,B 0,C 180,E1 -15135.792,E2 -15135.792} C_VEL
LIN {X 0,Y 429.326,Z 382.012,A -85,B 0,C 180,E1 -15137.344,E2 -15137.344} C_VEL
LIN {X 0,Y 430.756,Z 382.879,A -85,B 0,C 180,E1 -15137.983,E2 -15137.983} C_VEL
LIN {X 0,Y 432.894,Z 386.499,A -85,B 0,C 180,E1 -15139.007,E2 -15139.007} C_VEL
LIN {X 0,Y 436.387,Z 389.367,A -85,B 0,C 180,E1 -15140.417,E2 -15140.417} C_VEL
LIN {X 0,Y 439.091,Z 393.297,A -85,B 0,C 180,E1 -15141.508,E2 -15141.508} C_VEL
LIN {X 0,Y 441.913,Z 395.864,A -85,B 0,C 180,E1 -15142.517,E2 -15142.517} C_VEL
LIN {X 0,Y 445.097,Z 399.988,A -85,B 0,C 180,E1 -15143.64,E2 -15143.64} C_VEL
LIN {X 0,Y 450.118,Z 406.328,A -85,B 0,C 180,E1 -15145.281,E2 -15145.281} C_VEL
LIN {X 0,Y 454.628,Z 412.357,A -85,B 0,C 180,E1 -15146.658,E2 -15146.658} C_VEL
LIN {X 0,Y 460.709,Z 420.517,A -85,B 0,C 180,E1 -15148.379,E2 -15148.379} C_VEL
LIN {X 0,Y 471.19,Z 435.59,A -85,B 0,C 180,E1 -15151.077,E2 -15151.077} C_VEL
LIN {X 0,Y 482.617,Z 453.218,A -85,B 0,C 180,E1 -15153.71,E2 -15153.71} C_VEL
LIN {X 0,Y 493.474,Z 471.464,A -85,B 0,C 180,E1 -15155.987,E2 -15155.987} C_VEL
LIN {X 0,Y 499.53,Z 482.463,A -85,B 0,C 180,E1 -15157.184,E2 -15157.184} C_VEL
LIN {X 0,Y 487.311,Z 730.168,A -85,B 0,C 180,E1 -15161.029,E2 -15161.029} C_VEL
LIN {X 0,Y 485.219,Z 767,A -85,B 0,C 180,E1 -15161.641,E2 -15161.641} C_VEL
LIN {X 0,Y 482.763,Z 790.161,A -85,B 0,C 180,E1 -15162.175,E2 -15162.175} C_VEL
LIN {X 0,Y 479.68,Z 812.792,A -85,B 0,C 180,E1 -15162.854,E2 -15162.854} C_VEL
LIN {X 0,Y 475.653,Z 836.319,A -85,B 0,C 180,E1 -15163.773,E2 -15163.773} C_VEL
LIN {X 0,Y 471.762,Z 856.175,A -85,B 0,C 180,E1 -15164.722,E2 -15164.722} C_VEL
LIN {X 0,Y 466.5,Z 879.816,A -85,B 0,C 180,E1 -15166.093,E2 -15166.093} C_VEL
LIN {X 0,Y 461.785,Z 898.806,A -85,B 0,C 180,E1 -15167.408,E2 -15167.408} C_VEL
LIN {X 0,Y 456.132,Z 920.061,A -85,B 0,C 180,E1 -15169.137,E2 -15169.137} C_VEL
LIN {X 0,Y 450.707,Z 938.83,A -85,B 0,C 180,E1 -15170.946,E2 -15170.946} C_VEL
LIN {X 0,Y 445.06,Z 957.793,A -85,B 0,C 180,E1 -15173.06,E2 -15173.06} C_VEL
LIN {X 0,Y 439.664,Z 975.148,A -85,B 0,C 180,E1 -15175.35,E2 -15175.35} C_VEL
LIN {X 0,Y 434.536,Z 991.848,A -85,B 0,C 180,E1 -15177.89,E2 -15177.89} C_VEL
LIN {X 0,Y 429.874,Z 1006.94,A -85,B 0,C 180,E1 -15180.608,E2 -15180.608} C_VEL
LIN {X 0,Y 425.847,Z 1020.864,A -85,B 0,C 180,E1 -15183.505,E2 -15183.505} C_VEL
LIN {X 0,Y 422.601,Z 1032.668,A -85,B 0,C 180,E1 -15186.43,E2 -15186.43} C_VEL
LIN {X 0,Y 420.128,Z 1042.906,A -85,B 0,C 180,E1 -15189.376,E2 -15189.376} C_VEL
LIN {X 0,Y 418.201,Z 1052.212,A -85,B 0,C 180,E1 -15192.61,E2 -15192.61} C_VEL
LIN {X 0,Y 417.053,Z 1059.218,A -85,B 0,C 180,E1 -15195.561,E2 -15195.561} C_VEL
LIN {X 0,Y 416.287,Z 1065.785,A -85,B 0,C 180,E1 -15199.062,E2 -15199.062} C_VEL
LIN {X 0,Y 416.007,Z 1069.834,A -85,B 0,C 180,E1 -15201.999,E2 -15201.999} C_VEL
LIN {X 0,Y 415.95,Z 1072.645,A -85,B 0,C 180,E1 -15204.897,E2 -15204.897} C_VEL
LIN {X 0,Y 415.944,Z 1074.317,A -85,B 0,C 180,E1 -15208.209,E2 -15208.209} C_VEL
LIN {X 0,Y 415.954,Z 1074.456,A -85,B 0,C 180,E1 -15210.964,E2 -15210.964} C_VEL
LIN {X 0,Y 415.943,Z 1073.58,A -85,B 0,C 180,E1 -15213.583,E2 -15213.583} C_VEL
LIN {X 0,Y 415.958,Z 1071.358,A -85,B 0,C 180,E1 -15216.626,E2 -15216.626} C_VEL
LIN {X 0,Y 416.164,Z 1067.251,A -85,B 0,C 180,E1 -15219.962,E2 -15219.962} C_VEL
LIN {X 0,Y 416.61,Z 1062.575,A -85,B 0,C 180,E1 -15222.756,E2 -15222.756} C_VEL
LIN {X 0,Y 417.584,Z 1055.782,A -85,B 0,C 180,E1 -15225.984,E2 -15225.984} C_VEL
LIN {X 0,Y 419.143,Z 1047.327,A -85,B 0,C 180,E1 -15229.146,E2 -15229.146} C_VEL
LIN {X 0,Y 421.33,Z 1037.753,A -85,B 0,C 180,E1 -15232.169,E2 -15232.169} C_VEL
LIN {X 0,Y 424.356,Z 1026.061,A -85,B 0,C 180,E1 -15235.244,E2 -15235.244} C_VEL
LIN {X 0,Y 427.682,Z 1014.299,A -85,B 0,C 180,E1 -15237.903,E2 -15237.903} C_VEL
LIN {X 0,Y 432.351,Z 998.726,A -85,B 0,C 180,E1 -15240.906,E2 -15240.906} C_VEL
LIN {X 0,Y 436.58,Z 984.962,A -85,B 0,C 180,E1 -15243.187,E2 -15243.187} C_VEL
LIN {X 0,Y 442.06,Z 967.391,A -85,B 0,C 180,E1 -15245.706,E2 -15245.706} C_VEL
LIN {X 0,Y 447.038,Z 951.01,A -85,B 0,C 180,E1 -15247.715,E2 -15247.715} C_VEL
LIN {X 0,Y 452.531,Z 932.581,A -85,B 0,C 180,E1 -15249.684,E2 -15249.684} C_VEL
LIN {X 0,Y 458.075,Z 912.593,A -85,B 0,C 180,E1 -15251.489,E2 -15251.489} C_VEL
LIN {X 0,Y 463.203,Z 893.011,A -85,B 0,C 180,E1 -15253.01,E2 -15253.01} C_VEL
LIN {X 0,Y 468.442,Z 871.086,A -85,B 0,C 180,E1 -15254.436,E2 -15254.436} C_VEL
LIN {X 0,Y 472.77,Z 850.791,A -85,B 0,C 180,E1 -15255.545,E2 -15255.545} C_VEL
LIN {X 0,Y 477.305,Z 826.567,A -85,B 0,C 180,E1 -15256.629,E2 -15256.629} C_VEL
LIN {X 0,Y 480.752,Z 804.516,A -85,B 0,C 180,E1 -15257.406,E2 -15257.406} C_VEL
LIN {X 0,Y 483.879,Z 779.904,A -85,B 0,C 180,E1 -15258.076,E2 -15258.076} C_VEL
LIN {X 0,Y 485.863,Z 756.404,A -85,B 0,C 180,E1 -15258.54,E2 -15258.54} C_VEL
LIN {X 0,Y 497.86,Z 513.224,A -85,B 0,C 180,E1 -15262.33,E2 -15262.33} C_VEL
LIN {X 0,Y 499.35,Z 482.085,A -85,B 0,C 180,E1 -15262.827,E2 -15262.827} C_VEL
LIN {X 0,Y 488.571,Z 463.171,A -85,B 0,C 180,E1 -15264.984,E2 -15264.984} C_VEL
LIN {X 0,Y 479.452,Z 448.409,A -85,B 0,C 180,E1 -15266.951,E2 -15266.951} C_VEL
LIN {X 0,Y 470.156,Z 434.148,A -85,B 0,C 180,E1 -15269.131,E2 -15269.131} C_VEL
LIN {X 0,Y 460.248,Z 419.895,A -85,B 0,C 180,E1 -15271.696,E2 -15271.696} C_VEL
LIN {X 0,Y 452.227,Z 409.168,A -85,B 0,C 180,E1 -15274.002,E2 -15274.002} C_VEL
LIN {X 0,Y 447.264,Z 402.64,A -85,B 0,C 180,E1 -15275.57,E2 -15275.57} C_VEL
LIN {X 0,Y 444.102,Z 398.969,A -85,B 0,C 180,E1 -15276.62,E2 -15276.62} C_VEL
LIN {X 0,Y 441.304,Z 395.106,A -85,B 0,C 180,E1 -15277.626,E2 -15277.626} C_VEL
LIN {X 0,Y 437.766,Z 391.732,A -85,B 0,C 180,E1 -15278.916,E2 -15278.916} C_VEL
LIN {X 0,Y 436.118,Z 388.958,A -85,B 0,C 180,E1 -15279.605,E2 -15279.605} C_VEL
LIN {X 0,Y 432.829,Z 386.428,A -85,B 0,C 180,E1 -15280.92,E2 -15280.92} C_VEL
LIN {X 0,Y 430.743,Z 382.899,A -85,B 0,C 180,E1 -15281.912,E2 -15281.912} C_VEL
LIN {X 0,Y 426.831,Z 379.957,A -85,B 0,C 180,E1 -15283.743,E2 -15283.743} C_VEL
LIN {X 0,Y 425.001,Z 376.845,A -85,B 0,C 180,E1 -15284.792,E2 -15284.792} C_VEL
LIN {X 0,Y 424.713,Z 375.94,A -85,B 0,C 180,E1 -15284.991,E2 -15284.991} C_VEL
LIN {X 0,Y 421.236,Z 374.169,A -85,B 0,C 180,E1 -15286.968,E2 -15286.968} C_VEL
LIN {X 0,Y 419.097,Z 371.294,A -85,B 0,C 180,E1 -15288.509,E2 -15288.509} C_VEL
LIN {X 0,Y 418.507,Z 369.072,A -85,B 0,C 180,E1 -15289.12,E2 -15289.12} C_VEL
LIN {X 0,Y 418.488,Z 369.067,A -85,B 0,C 180,E1 -15292.863,E2 -15292.863} C_VEL
LIN {X 0,Y 418.486,Z 369.073,A -85,B 0,C 180,E1 -15296.576,E2 -15296.576} C_VEL
LIN {X 0,Y 418.494,Z 369.089,A -85,B 0,C 180,E1 -15300.411,E2 -15300.411} C_VEL
LIN {X 0,Y 418.515,Z 369.094,A -85,B 0,C 180,E1 -15304.11,E2 -15304.11} C_VEL
LIN {X 0,Y 418.534,Z 369.071,A -85,B 0,C 180,E1 -15307.965,E2 -15307.965} C_VEL
LIN {X 0,Y 418.533,Z 369.3,A -85,B 0,C 180,E1 -15311.36,E2 -15311.36} C_VEL
LIN {X 0,Y 419.58,Z 372.181,A -85,B 0,C 180,E1 -15312.296,E2 -15312.296} C_VEL
LIN {X 0,Y 421.874,Z 374.648,A -85,B 0,C 180,E1 -15313.85,E2 -15313.85} C_VEL
LIN {X 0,Y 424.82,Z 376.127,A -85,B 0,C 180,E1 -15315.494,E2 -15315.494} C_VEL
LIN {X 0,Y 426.343,Z 379.391,A -85,B 0,C 180,E1 -15316.421,E2 -15316.421} C_VEL
LIN {X 0,Y 429.092,Z 381.876,A -85,B 0,C 180,E1 -15317.774,E2 -15317.774} C_VEL
LIN {X 0,Y 430.742,Z 382.899,A -85,B 0,C 180,E1 -15318.508,E2 -15318.508} C_VEL
LIN {X 0,Y 432.982,Z 386.537,A -85,B 0,C 180,E1 -15319.564,E2 -15319.564} C_VEL
LIN {X 0,Y 436.493,Z 389.548,A -85,B 0,C 180,E1 -15320.973,E2 -15320.973} C_VEL
LIN {X 0,Y 439.226,Z 393.462,A -85,B 0,C 180,E1 -15322.063,E2 -15322.063} C_VEL
LIN {X 0,Y 441.815,Z 395.733,A -85,B 0,C 180,E1 -15322.979,E2 -15322.979} C_VEL
LIN {X 0,Y 444.911,Z 399.873,A -85,B 0,C 180,E1 -15324.073,E2 -15324.073} C_VEL
LIN {X 0,Y 447.033,Z 401.975,A -85,B 0,C 180,E1 -15324.761,E2 -15324.761} C_VEL
LIN {X 0,Y 450.675,Z 406.469,A -85,B 0,C 180,E1 -15325.918,E2 -15325.918} C_VEL
LIN {X 0,Y 452.601,Z 408.877,A -85,B 0,C 180,E1 -15326.504,E2 -15326.504} C_VEL
LIN {X 0,Y 457.102,Z 414.338,A -85,B 0,C 180,E1 -15327.806,E2 -15327.806} C_VEL
LIN {X 0,Y 462.528,Z 421.225,A -85,B 0,C 180,E1 -15329.282,E2 -15329.282} C_VEL
LIN {X 0,Y 470.338,Z 431.403,A -85,B 0,C 180,E1 -15331.247,E2 -15331.247} C_VEL
LIN {X 0,Y 480.133,Z 444.753,A -85,B 0,C 180,E1 -15333.496,E2 -15333.496} C_VEL
LIN {X 0,Y 491.349,Z 461.155,A -85,B 0,C 180,E1 -15335.843,E2 -15335.843} C_VEL
LIN {X 0,Y 499.651,Z 474.367,A -85,B 0,C 180,E1 -15337.459,E2 -15337.459} C_VEL
LIN {X 0,Y 487.078,Z 728.128,A -85,B 0,C 180,E1 -15341.395,E2 -15341.395} C_VEL
LIN {X 0,Y 485.241,Z 754.745,A -85,B 0,C 180,E1 -15341.88,E2 -15341.88} C_VEL
LIN {X 0,Y 482.919,Z 776.757,A -85,B 0,C 180,E1 -15342.427,E2 -15342.427} C_VEL
LIN {X 0,Y 479.469,Z 801.633,A -85,B 0,C 180,E1 -15343.254,E2 -15343.254} C_VEL
LIN {X 0,Y 476.09,Z 821.604,A -85,B 0,C 180,E1 -15344.088,E2 -15344.088} C_VEL
LIN {X 0,Y 471.613,Z 844.654,A -85,B 0,C 180,E1 -15345.26,E2 -15345.26} C_VEL
LIN {X 0,Y 467.017,Z 864.833,A -85,B 0,C 180,E1 -15346.502,E2 -15346.502} C_VEL
LIN {X 0,Y 461.884,Z 885.73,A -85,B 0,C 180,E1 -15348.016,E2 -15348.016} C_VEL
LIN {X 0,Y 456.404,Z 905.671,A -85,B 0,C 180,E1 -15349.738,E2 -15349.738} C_VEL
LIN {X 0,Y 451.306,Z 923.26,A -85,B 0,C 180,E1 -15351.496,E2 -15351.496} C_VEL
LIN {X 0,Y 445.438,Z 942.394,A -85,B 0,C 180,E1 -15353.738,E2 -15353.738} C_VEL
LIN {X 0,Y 440.72,Z 957.281,A -85,B 0,C 180,E1 -15355.761,E2 -15355.761} C_VEL
LIN {X 0,Y 435.334,Z 974.155,A -85,B 0,C 180,E1 -15358.421,E2 -15358.421} C_VEL
LIN {X 0,Y 431.116,Z 987.337,A -85,B 0,C 180,E1 -15360.853,E2 -15360.853} C_VEL
LIN {X 0,Y 426.917,Z 1001.011,A -85,B 0,C 180,E1 -15363.771,E2 -15363.771} C_VEL
LIN {X 0,Y 423.536,Z 1012.469,A -85,B 0,C 180,E1 -15366.688,E2 -15366.688} C_VEL
LIN {X 0,Y 420.764,Z 1023.05,A -85,B 0,C 180,E1 -15369.844,E2 -15369.844} C_VEL
LIN {X 0,Y 418.71,Z 1031.796,A -85,B 0,C 180,E1 -15373.062,E2 -15373.062} C_VEL
LIN {X 0,Y 417.355,Z 1039.019,A -85,B 0,C 180,E1 -15376.28,E2 -15376.28} C_VEL
LIN {X 0,Y 416.537,Z 1044.489,A -85,B 0,C 180,E1 -15379.488,E2 -15379.488} C_VEL
LIN {X 0,Y 416.179,Z 1048.077,A -85,B 0,C 180,E1 -15382.268,E2 -15382.268} C_VEL
LIN {X 0,Y 416.012,Z 1050.925,A -85,B 0,C 180,E1 -15385.451,E2 -15385.451} C_VEL
LIN {X 0,Y 415.957,Z 1052.186,A -85,B 0,C 180,E1 -15388.647,E2 -15388.647} C_VEL
LIN {X 0,Y 415.961,Z 1052.198,A -85,B 0,C 180,E1 -15391.378,E2 -15391.378} C_VEL
LIN {X 0,Y 415.978,Z 1051.54,A -85,B 0,C 180,E1 -15393.384,E2 -15393.384} C_VEL
LIN {X 0,Y 415.003,Z 1051.079,A -85,B 0,C 180,E1 -15394.443,E2 -15394.443} C_VEL
LIN {X 0,Y 408.669,Z 1048.903,A -85,B 0,C 180,E1 -15397.422,E2 -15397.422} C_VEL
LIN {X 0,Y 408.214,Z 1048.061,A -85,B 0,C 180,E1 -15398.194,E2 -15398.194} C_VEL
LIN {X 0,Y 408.696,Z 1044.037,A -85,B 0,C 180,E1 -15401.287,E2 -15401.287} C_VEL
LIN {X 0,Y 409.683,Z 1037.956,A -85,B 0,C 180,E1 -15404.704,E2 -15404.704} C_VEL
LIN {X 0,Y 411.093,Z 1031.215,A -85,B 0,C 180,E1 -15407.7,E2 -15407.7} C_VEL
LIN {X 0,Y 413.461,Z 1021.797,A -85,B 0,C 180,E1 -15411.121,E2 -15411.121} C_VEL
LIN {X 0,Y 416.284,Z 1011.826,A -85,B 0,C 180,E1 -15414.1,E2 -15414.1} C_VEL
LIN {X 0,Y 420.08,Z 999.654,A -85,B 0,C 180,E1 -15417.194,E2 -15417.194} C_VEL
LIN {X 0,Y 424.288,Z 986.635,A -85,B 0,C 180,E1 -15419.974,E2 -15419.974} C_VEL
LIN {X 0,Y 429.285,Z 971.795,A -85,B 0,C 180,E1 -15422.709,E2 -15422.709} C_VEL
LIN {X 0,Y 434.426,Z 956.269,A -85,B 0,C 180,E1 -15425.128,E2 -15425.128} C_VEL
LIN {X 0,Y 439.881,Z 939.753,A -85,B 0,C 180,E1 -15427.367,E2 -15427.367} C_VEL
LIN {X 0,Y 445.603,Z 921.468,A -85,B 0,C 180,E1 -15429.475,E2 -15429.475} C_VEL
LIN {X 0,Y 450.819,Z 904.098,A -85,B 0,C 180,E1 -15431.203,E2 -15431.203} C_VEL
LIN {X 0,Y 456.923,Z 882.147,A -85,B 0,C 180,E1 -15433.059,E2 -15433.059} C_VEL
LIN {X 0,Y 461.636,Z 863.499,A -85,B 0,C 180,E1 -15434.396,E2 -15434.396} C_VEL
LIN {X 0,Y 466.858,Z 840.833,A -85,B 0,C 180,E1 -15435.762,E2 -15435.762} C_VEL
LIN {X 0,Y 471.024,Z 819.587,A -85,B 0,C 180,E1 -15436.818,E2 -15436.818} C_VEL
LIN {X 0,Y 475.052,Z 795.897,A -85,B 0,C 180,E1 -15437.779,E2 -15437.779} C_VEL
LIN {X 0,Y 478.168,Z 772.412,A -85,B 0,C 180,E1 -15438.509,E2 -15438.509} C_VEL
LIN {X 0,Y 480.693,Z 747.809,A -85,B 0,C 180,E1 -15439.086,E2 -15439.086} C_VEL
LIN {X 0,Y 483.553,Z 695.326,A -85,B 0,C 180,E1 -15439.935,E2 -15439.935} C_VEL
LIN {X 0,Y 494.711,Z 478.149,A -85,B 0,C 180,E1 -15443.326,E2 -15443.326} C_VEL
LIN {X 0,Y 483.673,Z 460.957,A -85,B 0,C 180,E1 -15445.573,E2 -15445.573} C_VEL
LIN {X 0,Y 472.181,Z 444.466,A -85,B 0,C 180,E1 -15448.142,E2 -15448.142} C_VEL
LIN {X 0,Y 463.26,Z 432.53,A -85,B 0,C 180,E1 -15450.343,E2 -15450.343} C_VEL
LIN {X 0,Y 456.543,Z 423.812,A -85,B 0,C 180,E1 -15452.157,E2 -15452.157} C_VEL
LIN {X 0,Y 452.734,Z 419.024,A -85,B 0,C 180,E1 -15453.257,E2 -15453.257} C_VEL
LIN {X 0,Y 448.408,Z 413.667,A -85,B 0,C 180,E1 -15454.58,E2 -15454.58} C_VEL
LIN {X 0,Y 444.024,Z 408.294,A -85,B 0,C 180,E1 -15456.017,E2 -15456.017} C_VEL
LIN {X 0,Y 440.371,Z 404.04,A -85,B 0,C 180,E1 -15457.294,E2 -15457.294} C_VEL
LIN {X 0,Y 439.215,Z 402.509,A -85,B 0,C 180,E1 -15457.725,E2 -15457.725} C_VEL
LIN {X 0,Y 435.781,Z 398.941,A -85,B 0,C 180,E1 -15459.026,E2 -15459.026} C_VEL
LIN {X 0,Y 434.302,Z 396.582,A -85,B 0,C 180,E1 -15459.656,E2 -15459.656} C_VEL
LIN {X 0,Y 430.826,Z 393.516,A -85,B 0,C 180,E1 -15461.109,E2 -15461.109} C_VEL
LIN {X 0,Y 428.86,Z 390.242,A -85,B 0,C 180,E1 -15462.076,E2 -15462.076} C_VEL
LIN {X 0,Y 425.495,Z 387.858,A -85,B 0,C 180,E1 -15463.691,E2 -15463.691} C_VEL
LIN {X 0,Y 423.484,Z 384.464,A -85,B 0,C 180,E1 -15464.876,E2 -15464.876} C_VEL
LIN {X 0,Y 422.944,Z 383.636,A -85,B 0,C 180,E1 -15465.207,E2 -15465.207} C_VEL
LIN {X 0,Y 419.349,Z 381.402,A -85,B 0,C 180,E1 -15467.398,E2 -15467.398} C_VEL
LIN {X 0,Y 417.39,Z 377.975,A -85,B 0,C 180,E1 -15468.986,E2 -15468.986} C_VEL
LIN {X 0,Y 417.007,Z 376.93,A -85,B 0,C 180,E1 -15469.36,E2 -15469.36} C_VEL
LIN {X 0,Y 413.075,Z 374.967,A -85,B 0,C 180,E1 -15473.188,E2 -15473.188} C_VEL
LIN {X 0,Y 410.84,Z 371.334,A -85,B 0,C 180,E1 -15478.605,E2 -15478.605} C_VEL
LIN {X 0,Y 410.811,Z 371.306,A -85,B 0,C 180,E1 -15480.837,E2 -15480.837} C_VEL
LIN {X 0,Y 411.824,Z 373.448,A -85,B 0,C 180,E1 -15484.456,E2 -15484.456} C_VEL
LIN {X 0,Y 415.886,Z 376.655,A -85,B 0,C 180,E1 -15489.409,E2 -15489.409} C_VEL
LIN {X 0,Y 417.175,Z 377.23,A -85,B 0,C 180,E1 -15490.461,E2 -15490.461} C_VEL
LIN {X 0,Y 418.419,Z 380.185,A -85,B 0,C 180,E1 -15491.58,E2 -15491.58} C_VEL
LIN {X 0,Y 421.394,Z 382.985,A -85,B 0,C 180,E1 -15493.586,E2 -15493.586} C_VEL
LIN {X 0,Y 423.249,Z 383.981,A -85,B 0,C 180,E1 -15494.642,E2 -15494.642} C_VEL
LIN {X 0,Y 425.103,Z 387.341,A -85,B 0,C 180,E1 -15495.764,E2 -15495.764} C_VEL
LIN {X 0,Y 428.386,Z 390.039,A -85,B 0,C 180,E1 -15497.383,E2 -15497.383} C_VEL
LIN {X 0,Y 429.14,Z 390.75,A -85,B 0,C 180,E1 -15497.737,E2 -15497.737} C_VEL
LIN {X 0,Y 431.635,Z 394.517,A -85,B 0,C 180,E1 -15498.924,E2 -15498.924} C_VEL
LIN {X 0,Y 434.626,Z 397.081,A -85,B 0,C 180,E1 -15500.152,E2 -15500.152} C_VEL
LIN {X 0,Y 437.639,Z 401.168,A -85,B 0,C 180,E1 -15501.372,E2 -15501.372} C_VEL
LIN {X 0,Y 439.92,Z 403.293,A -85,B 0,C 180,E1 -15502.202,E2 -15502.202} C_VEL
LIN {X 0,Y 443.424,Z 407.703,A -85,B 0,C 180,E1 -15503.453,E2 -15503.453} C_VEL
LIN {X 0,Y 448.011,Z 413.753,A -85,B 0,C 180,E1 -15504.985,E2 -15504.985} C_VEL
LIN {X 0,Y 452.561,Z 419.934,A -85,B 0,C 180,E1 -15506.401,E2 -15506.401} C_VEL
LIN {X 0,Y 458.165,Z 427.56,A -85,B 0,C 180,E1 -15508.019,E2 -15508.019} C_VEL
LIN {X 0,Y 468.397,Z 442.51,A -85,B 0,C 180,E1 -15510.713,E2 -15510.713} C_VEL
LIN {X 0,Y 479.328,Z 459.628,A -85,B 0,C 180,E1 -15513.291,E2 -15513.291} C_VEL
LIN {X 0,Y 489.859,Z 477.561,A -85,B 0,C 180,E1 -15515.555,E2 -15515.555} C_VEL
LIN {X 0,Y 494.506,Z 486.197,A -85,B 0,C 180,E1 -15516.503,E2 -15516.503} C_VEL
LIN {X 0,Y 481.836,Z 734.899,A -85,B 0,C 180,E1 -15520.386,E2 -15520.386} C_VEL
LIN {X 0,Y 479.757,Z 768.426,A -85,B 0,C 180,E1 -15520.959,E2 -15520.959} C_VEL
LIN {X 0,Y 477.319,Z 790.611,A -85,B 0,C 180,E1 -15521.477,E2 -15521.477} C_VEL
LIN {X 0,Y 474.014,Z 814.068,A -85,B 0,C 180,E1 -15522.189,E2 -15522.189} C_VEL
LIN {X 0,Y 469.974,Z 836.741,A -85,B 0,C 180,E1 -15523.089,E2 -15523.089} C_VEL
LIN {X 0,Y 465.942,Z 856.679,A -85,B 0,C 180,E1 -15524.051,E2 -15524.051} C_VEL
LIN {X 0,Y 460.42,Z 880.599,A -85,B 0,C 180,E1 -15525.456,E2 -15525.456} C_VEL
LIN {X 0,Y 455.779,Z 898.682,A -85,B 0,C 180,E1 -15526.72,E2 -15526.72} C_VEL
LIN {X 0,Y 449.983,Z 919.785,A -85,B 0,C 180,E1 -15528.449,E2 -15528.449} C_VEL
LIN {X 0,Y 444.352,Z 938.614,A -85,B 0,C 180,E1 -15530.278,E2 -15530.278} C_VEL
LIN {X 0,Y 438.523,Z 957.489,A -85,B 0,C 180,E1 -15532.401,E2 -15532.401} C_VEL
LIN {X 0,Y 432.879,Z 974.93,A -85,B 0,C 180,E1 -15534.727,E2 -15534.727} C_VEL
LIN {X 0,Y 427.538,Z 991.629,A -85,B 0,C 180,E1 -15537.3,E2 -15537.3} C_VEL
LIN {X 0,Y 422.664,Z 1006.721,A -85,B 0,C 180,E1 -15540.055,E2 -15540.055} C_VEL
LIN {X 0,Y 418.44,Z 1020.644,A -85,B 0,C 180,E1 -15542.998,E2 -15542.998} C_VEL
LIN {X 0,Y 415.019,Z 1032.449,A -85,B 0,C 180,E1 -15545.973,E2 -15545.973} C_VEL
LIN {X 0,Y 412.406,Z 1042.71,A -85,B 0,C 180,E1 -15548.979,E2 -15548.979} C_VEL
LIN {X 0,Y 410.339,Z 1052.127,A -85,B 0,C 180,E1 -15552.321,E2 -15552.321} C_VEL
LIN {X 0,Y 409.139,Z 1059,A -85,B 0,C 180,E1 -15555.276,E2 -15555.276} C_VEL
LIN {X 0,Y 408.319,Z 1065.569,A -85,B 0,C 180,E1 -15558.845,E2 -15558.845} C_VEL
LIN {X 0,Y 408.02,Z 1069.605,A -85,B 0,C 180,E1 -15561.829,E2 -15561.829} C_VEL
LIN {X 0,Y 407.951,Z 1072.43,A -85,B 0,C 180,E1 -15564.797,E2 -15564.797} C_VEL
LIN {X 0,Y 407.946,Z 1074.104,A -85,B 0,C 180,E1 -15568.174,E2 -15568.174} C_VEL
LIN {X 0,Y 407.957,Z 1074.243,A -85,B 0,C 180,E1 -15570.983,E2 -15570.983} C_VEL
LIN {X 0,Y 407.944,Z 1073.365,A -85,B 0,C 180,E1 -15573.654,E2 -15573.654} C_VEL
LIN {X 0,Y 407.959,Z 1071.259,A -85,B 0,C 180,E1 -15576.615,E2 -15576.615} C_VEL
LIN {X 0,Y 408.169,Z 1067.245,A -85,B 0,C 180,E1 -15580.016,E2 -15580.016} C_VEL
LIN {X 0,Y 408.632,Z 1062.616,A -85,B 0,C 180,E1 -15582.866,E2 -15582.866} C_VEL
LIN {X 0,Y 409.59,Z 1056.199,A -85,B 0,C 180,E1 -15586.013,E2 -15586.013} C_VEL
LIN {X 0,Y 411.284,Z 1047.491,A -85,B 0,C 180,E1 -15589.389,E2 -15589.389} C_VEL
LIN {X 0,Y 413.432,Z 1038.463,A -85,B 0,C 180,E1 -15592.315,E2 -15592.315} C_VEL
LIN {X 0,Y 416.707,Z 1026.42,A -85,B 0,C 180,E1 -15595.589,E2 -15595.589} C_VEL
LIN {X 0,Y 420.175,Z 1014.692,A -85,B 0,C 180,E1 -15598.298,E2 -15598.298} C_VEL
LIN {X 0,Y 425.032,Z 999.213,A -85,B 0,C 180,E1 -15601.355,E2 -15601.355} C_VEL
LIN {X 0,Y 429.67,Z 984.739,A -85,B 0,C 180,E1 -15603.792,E2 -15603.792} C_VEL
LIN {X 0,Y 435.367,Z 967.195,A -85,B 0,C 180,E1 -15606.337,E2 -15606.337} C_VEL
LIN {X 0,Y 440.485,Z 950.977,A -85,B 0,C 180,E1 -15608.349,E2 -15608.349} C_VEL
LIN {X 0,Y 446.303,Z 932.128,A -85,B 0,C 180,E1 -15610.383,E2 -15610.383} C_VEL
LIN {X 0,Y 452.172,Z 911.631,A -85,B 0,C 180,E1 -15612.24,E2 -15612.24} C_VEL
LIN {X 0,Y 457.71,Z 891.157,A -85,B 0,C 180,E1 -15613.828,E2 -15613.828} C_VEL
LIN {X 0,Y 462.899,Z 869.854,A -85,B 0,C 180,E1 -15615.201,E2 -15615.201} C_VEL
LIN {X 0,Y 467.368,Z 849.434,A -85,B 0,C 180,E1 -15616.312,E2 -15616.312} C_VEL
LIN {X 0,Y 472.119,Z 824.402,A -85,B 0,C 180,E1 -15617.416,E2 -15617.416} C_VEL
LIN {X 0,Y 475.57,Z 802.717,A -85,B 0,C 180,E1 -15618.171,E2 -15618.171} C_VEL
LIN {X 0,Y 478.878,Z 776.322,A -85,B 0,C 180,E1 -15618.864,E2 -15618.864} C_VEL
LIN {X 0,Y 480.723,Z 754.023,A -85,B 0,C 180,E1 -15619.295,E2 -15619.295} C_VEL
LIN {X 0,Y 493.306,Z 506.927,A -85,B 0,C 180,E1 -15623.164,E2 -15623.164} C_VEL
LIN {X 0,Y 494.325,Z 485.724,A -85,B 0,C 180,E1 -15623.51,E2 -15623.51} C_VEL
LIN {X 0,Y 483.923,Z 467.43,A -85,B 0,C 180,E1 -15625.662,E2 -15625.662} C_VEL
LIN {X 0,Y 475.048,Z 452.909,A -85,B 0,C 180,E1 -15627.646,E2 -15627.646} C_VEL
LIN {X 0,Y 466.048,Z 439.17,A -85,B 0,C 180,E1 -15629.829,E2 -15629.829} C_VEL
LIN {X 0,Y 457.399,Z 426.504,A -85,B 0,C 180,E1 -15632.143,E2 -15632.143} C_VEL
LIN {X 0,Y 449.71,Z 416.077,A -85,B 0,C 180,E1 -15634.412,E2 -15634.412} C_VEL
LIN {X 0,Y 445.016,Z 409.783,A -85,B 0,C 180,E1 -15635.933,E2 -15635.933} C_VEL
LIN {X 0,Y 439.736,Z 403.015,A -85,B 0,C 180,E1 -15637.788,E2 -15637.788} C_VEL
LIN {X 0,Y 435.61,Z 398.766,A -85,B 0,C 180,E1 -15639.334,E2 -15639.334} C_VEL
LIN {X 0,Y 434.202,Z 396.496,A -85,B 0,C 180,E1 -15639.933,E2 -15639.933} C_VEL
LIN {X 0,Y 430.849,Z 393.62,A -85,B 0,C 180,E1 -15641.321,E2 -15641.321} C_VEL
LIN {X 0,Y 428.725,Z 390.213,A -85,B 0,C 180,E1 -15642.35,E2 -15642.35} C_VEL
LIN {X 0,Y 425.484,Z 387.788,A -85,B 0,C 180,E1 -15643.901,E2 -15643.901} C_VEL
LIN {X 0,Y 423.384,Z 384.381,A -85,B 0,C 180,E1 -15645.118,E2 -15645.118} C_VEL
LIN {X 0,Y 423.019,Z 383.652,A -85,B 0,C 180,E1 -15645.35,E2 -15645.35} C_VEL
LIN {X 0,Y 419.86,Z 381.871,A -85,B 0,C 180,E1 -15647.204,E2 -15647.204} C_VEL
LIN {X 0,Y 417.689,Z 378.838,A -85,B 0,C 180,E1 -15648.819,E2 -15648.819} C_VEL
LIN {X 0,Y 416.962,Z 376.921,A -85,B 0,C 180,E1 -15649.499,E2 -15649.499} C_VEL
LIN {X 0,Y 413.043,Z 374.909,A -85,B 0,C 180,E1 -15653.188,E2 -15653.188} C_VEL
LIN {X 0,Y 410.58,Z 370.081,A -85,B 0,C 180,E1 -15659.39,E2 -15659.39} C_VEL
LIN {X 0,Y 410.651,Z 370.459,A -85,B 0,C 180,E1 -15661.814,E2 -15661.814} C_VEL
LIN {X 0,Y 414.827,Z 376.213,A -85,B 0,C 180,E1 -15669.154,E2 -15669.154} C_VEL
LIN {X 0,Y 417.162,Z 377.189,A -85,B 0,C 180,E1 -15671.09,E2 -15671.09} C_VEL
LIN {X 0,Y 418.702,Z 380.605,A -85,B 0,C 180,E1 -15672.411,E2 -15672.411} C_VEL
LIN {X 0,Y 421.818,Z 383.197,A -85,B 0,C 180,E1 -15674.412,E2 -15674.412} C_VEL
LIN {X 0,Y 423.296,Z 384.035,A -85,B 0,C 180,E1 -15675.236,E2 -15675.236} C_VEL
LIN {X 0,Y 425.233,Z 387.555,A -85,B 0,C 180,E1 -15676.39,E2 -15676.39} C_VEL
LIN {X 0,Y 428.438,Z 390.061,A -85,B 0,C 180,E1 -15677.943,E2 -15677.943} C_VEL
LIN {X 0,Y 429.126,Z 390.75,A -85,B 0,C 180,E1 -15678.264,E2 -15678.264} C_VEL
LIN {X 0,Y 431.723,Z 394.563,A -85,B 0,C 180,E1 -15679.482,E2 -15679.482} C_VEL
LIN {X 0,Y 434.655,Z 397.13,A -85,B 0,C 180,E1 -15680.678,E2 -15680.678} C_VEL
LIN {X 0,Y 437.607,Z 401.172,A -85,B 0,C 180,E1 -15681.866,E2 -15681.866} C_VEL
LIN {X 0,Y 439.899,Z 403.315,A -85,B 0,C 180,E1 -15682.696,E2 -15682.696} C_VEL
LIN {X 0,Y 443.42,Z 407.767,A -85,B 0,C 180,E1 -15683.947,E2 -15683.947} C_VEL
LIN {X 0,Y 445.051,Z 409.553,A -85,B 0,C 180,E1 -15684.489,E2 -15684.489} C_VEL
LIN {X 0,Y 448.956,Z 414.195,A -85,B 0,C 180,E1 -15685.74,E2 -15685.74} C_VEL
LIN {X 0,Y 455.11,Z 422.051,A -85,B 0,C 180,E1 -15687.583,E2 -15687.583} C_VEL
LIN {X 0,Y 461.996,Z 430.756,A -85,B 0,C 180,E1 -15689.461,E2 -15689.461} C_VEL
LIN {X 0,Y 472.909,Z 445.543,A -85,B 0,C 180,E1 -15692.16,E2 -15692.16} C_VEL
LIN {X 0,Y 484.242,Z 461.885,A -85,B 0,C 180,E1 -15694.672,E2 -15694.672} C_VEL
LIN {X 0,Y 494.632,Z 478.104,A -85,B 0,C 180,E1 -15696.777,E2 -15696.777} C_VEL
LIN {X 0,Y 481.715,Z 730.598,A -85,B 0,C 180,E1 -15700.716,E2 -15700.716} C_VEL
LIN {X 0,Y 479.857,Z 755.794,A -85,B 0,C 180,E1 -15701.186,E2 -15701.186} C_VEL
LIN {X 0,Y 477.38,Z 778.478,A -85,B 0,C 180,E1 -15701.76,E2 -15701.76} C_VEL
LIN {X 0,Y 473.881,Z 802.595,A -85,B 0,C 180,E1 -15702.575,E2 -15702.575} C_VEL
LIN {X 0,Y 470.296,Z 823.106,A -85,B 0,C 180,E1 -15703.443,E2 -15703.443} C_VEL
LIN {X 0,Y 465.227,Z 847.876,A -85,B 0,C 180,E1 -15704.739,E2 -15704.739} C_VEL
LIN {X 0,Y 460.691,Z 867.092,A -85,B 0,C 180,E1 -15705.948,E2 -15705.948} C_VEL
LIN {X 0,Y 455.011,Z 889.093,A -85,B 0,C 180,E1 -15707.592,E2 -15707.592} C_VEL
LIN {X 0,Y 449.836,Z 907.219,A -85,B 0,C 180,E1 -15709.194,E2 -15709.194} C_VEL
LIN {X 0,Y 444.242,Z 925.897,A -85,B 0,C 180,E1 -15711.1,E2 -15711.1} C_VEL
LIN {X 0,Y 438.371,Z 944.123,A -85,B 0,C 180,E1 -15713.302,E2 -15713.302} C_VEL
LIN {X 0,Y 433.079,Z 960.253,A -85,B 0,C 180,E1 -15715.552,E2 -15715.552} C_VEL
LIN {X 0,Y 427.836,Z 975.901,A -85,B 0,C 180,E1 -15718.117,E2 -15718.117} C_VEL
LIN {X 0,Y 423.481,Z 989.027,A -85,B 0,C 180,E1 -15720.605,E2 -15720.605} C_VEL
LIN {X 0,Y 418.874,Z 1003.324,A -85,B 0,C 180,E1 -15723.793,E2 -15723.793} C_VEL
LIN {X 0,Y 415.62,Z 1014.024,A -85,B 0,C 180,E1 -15726.612,E2 -15726.612} C_VEL
LIN {X 0,Y 412.568,Z 1025.113,A -85,B 0,C 180,E1 -15730.111,E2 -15730.111} C_VEL
LIN {X 0,Y 410.714,Z 1032.894,A -85,B 0,C 180,E1 -15733.092,E2 -15733.092} C_VEL
LIN {X 0,Y 409.227,Z 1040.512,A -85,B 0,C 180,E1 -15736.722,E2 -15736.722} C_VEL
LIN {X 0,Y 408.512,Z 1045.334,A -85,B 0,C 180,E1 -15739.723,E2 -15739.723} C_VEL
LIN {X 0,Y 408.127,Z 1049.366,A -85,B 0,C 180,E1 -15743.105,E2 -15743.105} C_VEL
LIN {X 0,Y 407.99,Z 1051.611,A -85,B 0,C 180,E1 -15746.347,E2 -15746.347} C_VEL
LIN {X 0,Y 407.958,Z 1052.484,A -85,B 0,C 180,E1 -15749.158,E2 -15749.158} C_VEL
LIN {X 0,Y 407.973,Z 1052.252,A -85,B 0,C 180,E1 -15752.388,E2 -15752.388} C_VEL
LIN {X 0,Y 408.043,Z 1050.443,A -85,B 0,C 180,E1 -15755.625,E2 -15755.625} C_VEL
LIN {X 0,Y 408.214,Z 1048.061,A -85,B 0,C 180,E1 -15758.194,E2 -15758.194} C_VEL
LIN {X 0,Y 407.358,Z 1046.942,A -85,B 0,C 180,E1 -15759.265,E2 -15759.265} C_VEL
LIN {X 0,Y 401.553,Z 1043.163,A -85,B 0,C 180,E1 -15762.202,E2 -15762.202} C_VEL
LIN {X 0,Y 401.148,Z 1041.744,A -85,B 0,C 180,E1 -15763.054,E2 -15763.054} C_VEL
LIN {X 0,Y 402.389,Z 1035.496,A -85,B 0,C 180,E1 -15766.308,E2 -15766.308} C_VEL
LIN {X 0,Y 404.35,Z 1027.344,A -85,B 0,C 180,E1 -15769.652,E2 -15769.652} C_VEL
LIN {X 0,Y 406.729,Z 1018.851,A -85,B 0,C 180,E1 -15772.551,E2 -15772.551} C_VEL
LIN {X 0,Y 410.496,Z 1006.745,A -85,B 0,C 180,E1 -15776.005,E2 -15776.005} C_VEL
LIN {X 0,Y 414.232,Z 995.483,A -85,B 0,C 180,E1 -15778.709,E2 -15778.709} C_VEL
LIN {X 0,Y 419.178,Z 981.194,A -85,B 0,C 180,E1 -15781.653,E2 -15781.653} C_VEL
LIN {X 0,Y 424.172,Z 966.789,A -85,B 0,C 180,E1 -15784.167,E2 -15784.167} C_VEL
LIN {X 0,Y 429.818,Z 950.576,A -85,B 0,C 180,E1 -15786.623,E2 -15786.623} C_VEL
LIN {X 0,Y 435.69,Z 932.92,A -85,B 0,C 180,E1 -15788.879,E2 -15788.879} C_VEL
LIN {X 0,Y 441.755,Z 914.215,A -85,B 0,C 180,E1 -15790.94,E2 -15790.94} C_VEL
LIN {X 0,Y 447.631,Z 894.469,A -85,B 0,C 180,E1 -15792.77,E2 -15792.77} C_VEL
LIN {X 0,Y 453.017,Z 875.096,A -85,B 0,C 180,E1 -15794.313,E2 -15794.313} C_VEL
LIN {X 0,Y 458.451,Z 853.339,A -85,B 0,C 180,E1 -15795.763,E2 -15795.763} C_VEL
LIN {X 0,Y 462.69,Z 834.32,A -85,B 0,C 180,E1 -15796.832,E2 -15796.832} C_VEL
LIN {X 0,Y 467.189,Z 811.27,A -85,B 0,C 180,E1 -15797.913,E2 -15797.913} C_VEL
LIN {X 0,Y 470.661,Z 789.502,A -85,B 0,C 180,E1 -15798.722,E2 -15798.722} C_VEL
LIN {X 0,Y 473.63,Z 766.884,A -85,B 0,C 180,E1 -15799.389,E2 -15799.389} C_VEL
LIN {X 0,Y 475.897,Z 742.012,A -85,B 0,C 180,E1 -15799.92,E2 -15799.92} C_VEL
LIN {X 0,Y 488.436,Z 506.769,A -85,B 0,C 180,E1 -15803.629,E2 -15803.629} C_VEL
LIN {X 0,Y 489.683,Z 482.013,A -85,B 0,C 180,E1 -15804.034,E2 -15804.034} C_VEL
LIN {X 0,Y 479.175,Z 465.536,A -85,B 0,C 180,E1 -15806.249,E2 -15806.249} C_VEL
LIN {X 0,Y 468.574,Z 450.296,A -85,B 0,C 180,E1 -15808.694,E2 -15808.694} C_VEL
LIN {X 0,Y 458.786,Z 436.894,A -85,B 0,C 180,E1 -15811.206,E2 -15811.206} C_VEL
LIN {X 0,Y 450.59,Z 426.388,A -85,B 0,C 180,E1 -15813.546,E2 -15813.546} C_VEL
LIN {X 0,Y 445.939,Z 420.65,A -85,B 0,C 180,E1 -15814.997,E2 -15814.997} C_VEL
LIN {X 0,Y 441.809,Z 415.52,A -85,B 0,C 180,E1 -15816.385,E2 -15816.385} C_VEL
LIN {X 0,Y 438.07,Z 410.927,A -85,B 0,C 180,E1 -15817.735,E2 -15817.735} C_VEL
LIN {X 0,Y 433.507,Z 405.742,A -85,B 0,C 180,E1 -15819.512,E2 -15819.512} C_VEL
LIN {X 0,Y 432.251,Z 403.994,A -85,B 0,C 180,E1 -15820.05,E2 -15820.05} C_VEL
LIN {X 0,Y 428.744,Z 400.514,A -85,B 0,C 180,E1 -15821.578,E2 -15821.578} C_VEL
LIN {X 0,Y 427.063,Z 397.859,A -85,B 0,C 180,E1 -15822.42,E2 -15822.42} C_VEL
LIN {X 0,Y 423.797,Z 395.265,A -85,B 0,C 180,E1 -15824.046,E2 -15824.046} C_VEL
LIN {X 0,Y 421.516,Z 391.441,A -85,B 0,C 180,E1 -15825.437,E2 -15825.437} C_VEL
LIN {X 0,Y 418,Z 389.099,A -85,B 0,C 180,E1 -15827.638,E2 -15827.638} C_VEL
LIN {X 0,Y 415.98,Z 385.44,A -85,B 0,C 180,E1 -15829.334,E2 -15829.334} C_VEL
LIN {X 0,Y 415.697,Z 384.8,A -85,B 0,C 180,E1 -15829.607,E2 -15829.607} C_VEL
LIN {X 0,Y 411.801,Z 382.65,A -85,B 0,C 180,E1 -15833.587,E2 -15833.587} C_VEL
LIN {X 0,Y 409.847,Z 379.253,A -85,B 0,C 180,E1 -15838.742,E2 -15838.742} C_VEL
LIN {X 0,Y 409.835,Z 379.262,A -85,B 0,C 180,E1 -15840.839,E2 -15840.839} C_VEL
LIN {X 0,Y 410.846,Z 381.441,A -85,B 0,C 180,E1 -15844.467,E2 -15844.467} C_VEL
LIN {X 0,Y 414.922,Z 384.609,A -85,B 0,C 180,E1 -15849.432,E2 -15849.432} C_VEL
LIN {X 0,Y 415.862,Z 385.085,A -85,B 0,C 180,E1 -15850.214,E2 -15850.214} C_VEL
LIN {X 0,Y 417.348,Z 388.242,A -85,B 0,C 180,E1 -15851.54,E2 -15851.54} C_VEL
LIN {X 0,Y 420.439,Z 390.984,A -85,B 0,C 180,E1 -15853.618,E2 -15853.618} C_VEL
LIN {X 0,Y 421.755,Z 391.754,A -85,B 0,C 180,E1 -15854.379,E2 -15854.379} C_VEL
LIN {X 0,Y 423.887,Z 395.315,A -85,B 0,C 180,E1 -15855.67,E2 -15855.67} C_VEL
LIN {X 0,Y 427.481,Z 398.409,A -85,B 0,C 180,E1 -15857.457,E2 -15857.457} C_VEL
LIN {X 0,Y 430.235,Z 402.359,A -85,B 0,C 180,E1 -15858.777,E2 -15858.777} C_VEL
LIN {X 0,Y 432.808,Z 404.617,A -85,B 0,C 180,E1 -15859.853,E2 -15859.853} C_VEL
LIN {X 0,Y 436.027,Z 408.867,A -85,B 0,C 180,E1 -15861.173,E2 -15861.173} C_VEL
LIN {X 0,Y 438.022,Z 410.833,A -85,B 0,C 180,E1 -15861.915,E2 -15861.915} C_VEL
LIN {X 0,Y 445.113,Z 419.941,A -85,B 0,C 180,E1 -15864.414,E2 -15864.414} C_VEL
LIN {X 0,Y 453.535,Z 431.567,A -85,B 0,C 180,E1 -15867.043,E2 -15867.043} C_VEL
LIN {X 0,Y 461.851,Z 443.748,A -85,B 0,C 180,E1 -15869.365,E2 -15869.365} C_VEL
LIN {X 0,Y 470.723,Z 457.483,A -85,B 0,C 180,E1 -15871.61,E2 -15871.61} C_VEL
LIN {X 0,Y 479.232,Z 471.361,A -85,B 0,C 180,E1 -15873.585,E2 -15873.585} C_VEL
LIN {X 0,Y 489.561,Z 489.614,A -85,B 0,C 180,E1 -15875.802,E2 -15875.802} C_VEL
LIN {X 0,Y 476.728,Z 733.588,A -85,B 0,C 180,E1 -15879.633,E2 -15879.633} C_VEL
LIN {X 0,Y 474.581,Z 767.739,A -85,B 0,C 180,E1 -15880.216,E2 -15880.216} C_VEL
LIN {X 0,Y 472.048,Z 790.278,A -85,B 0,C 180,E1 -15880.742,E2 -15880.742} C_VEL
LIN {X 0,Y 468.64,Z 813.862,A -85,B 0,C 180,E1 -15881.459,E2 -15881.459} C_VEL
LIN {X 0,Y 464.489,Z 836.524,A -85,B 0,C 180,E1 -15882.36,E2 -15882.36} C_VEL
LIN {X 0,Y 460.185,Z 857.191,A -85,B 0,C 180,E1 -15883.362,E2 -15883.362} C_VEL
LIN {X 0,Y 454.654,Z 880.387,A -85,B 0,C 180,E1 -15884.736,E2 -15884.736} C_VEL
LIN {X 0,Y 449.647,Z 899.284,A -85,B 0,C 180,E1 -15886.068,E2 -15886.068} C_VEL
LIN {X 0,Y 443.375,Z 921.195,A -85,B 0,C 180,E1 -15887.898,E2 -15887.898} C_VEL
LIN {X 0,Y 437.867,Z 939.011,A -85,B 0,C 180,E1 -15889.655,E2 -15889.655} C_VEL
LIN {X 0,Y 431.81,Z 957.87,A -85,B 0,C 180,E1 -15891.811,E2 -15891.811} C_VEL
LIN {X 0,Y 426.15,Z 974.711,A -85,B 0,C 180,E1 -15894.085,E2 -15894.085} C_VEL
LIN {X 0,Y 420.586,Z 991.41,A -85,B 0,C 180,E1 -15896.69,E2 -15896.69} C_VEL
LIN {X 0,Y 415.494,Z 1006.501,A -85,B 0,C 180,E1 -15899.484,E2 -15899.484} C_VEL
LIN {X 0,Y 411.064,Z 1020.425,A -85,B 0,C 180,E1 -15902.473,E2 -15902.473} C_VEL
LIN {X 0,Y 407.37,Z 1032.565,A -85,B 0,C 180,E1 -15905.592,E2 -15905.592} C_VEL
LIN {X 0,Y 404.492,Z 1043.395,A -85,B 0,C 180,E1 -15908.844,E2 -15908.844} C_VEL
LIN {X 0,Y 402.39,Z 1052.494,A -85,B 0,C 180,E1 -15912.203,E2 -15912.203} C_VEL
LIN {X 0,Y 401.093,Z 1059.709,A -85,B 0,C 180,E1 -15915.417,E2 -15915.417} C_VEL
LIN {X 0,Y 400.307,Z 1065.775,A -85,B 0,C 180,E1 -15918.911,E2 -15918.911} C_VEL
LIN {X 0,Y 400.02,Z 1069.575,A -85,B 0,C 180,E1 -15921.828,E2 -15921.828} C_VEL
LIN {X 0,Y 399.951,Z 1072.448,A -85,B 0,C 180,E1 -15924.98,E2 -15924.98} C_VEL
LIN {X 0,Y 399.949,Z 1073.914,A -85,B 0,C 180,E1 -15928.281,E2 -15928.281} C_VEL
LIN {X 0,Y 399.959,Z 1074.029,A -85,B 0,C 180,E1 -15931.003,E2 -15931.003} C_VEL
LIN {X 0,Y 399.945,Z 1073.151,A -85,B 0,C 180,E1 -15933.727,E2 -15933.727} C_VEL
LIN {X 0,Y 399.963,Z 1071.044,A -85,B 0,C 180,E1 -15936.748,E2 -15936.748} C_VEL
LIN {X 0,Y 400.187,Z 1067.028,A -85,B 0,C 180,E1 -15940.218,E2 -15940.218} C_VEL
LIN {X 0,Y 400.687,Z 1062.398,A -85,B 0,C 180,E1 -15943.125,E2 -15943.125} C_VEL
LIN {X 0,Y 401.715,Z 1055.98,A -85,B 0,C 180,E1 -15946.335,E2 -15946.335} C_VEL
LIN {X 0,Y 403.468,Z 1047.497,A -85,B 0,C 180,E1 -15949.697,E2 -15949.697} C_VEL
LIN {X 0,Y 405.662,Z 1038.707,A -85,B 0,C 180,E1 -15952.613,E2 -15952.613} C_VEL
LIN {X 0,Y 409.242,Z 1026.197,A -85,B 0,C 180,E1 -15956.09,E2 -15956.09} C_VEL
LIN {X 0,Y 412.844,Z 1014.604,A -85,B 0,C 180,E1 -15958.814,E2 -15958.814} C_VEL
LIN {X 0,Y 417.739,Z 999.701,A -85,B 0,C 180,E1 -15961.818,E2 -15961.818} C_VEL
LIN {X 0,Y 422.521,Z 985.369,A -85,B 0,C 180,E1 -15964.279,E2 -15964.279} C_VEL
LIN {X 0,Y 428.244,Z 968.524,A -85,B 0,C 180,E1 -15966.787,E2 -15966.787} C_VEL
LIN {X 0,Y 433.928,Z 951.123,A -85,B 0,C 180,E1 -15968.981,E2 -15968.981} C_VEL
LIN {X 0,Y 439.6,Z 933.36,A -85,B 0,C 180,E1 -15970.925,E2 -15970.925} C_VEL
LIN {X 0,Y 445.721,Z 912.887,A -85,B 0,C 180,E1 -15972.822,E2 -15972.822} C_VEL
LIN {X 0,Y 450.949,Z 894.197,A -85,B 0,C 180,E1 -15974.303,E2 -15974.303} C_VEL
LIN {X 0,Y 456.972,Z 870.641,A -85,B 0,C 180,E1 -15975.864,E2 -15975.864} C_VEL
LIN {X 0,Y 461.558,Z 850.348,A -85,B 0,C 180,E1 -15976.982,E2 -15976.982} C_VEL
LIN {X 0,Y 466.487,Z 825.377,A -85,B 0,C 180,E1 -15978.1,E2 -15978.1} C_VEL
LIN {X 0,Y 470.076,Z 803.547,A -85,B 0,C 180,E1 -15978.869,E2 -15978.869} C_VEL
LIN {X 0,Y 473.44,Z 777.98,A -85,B 0,C 180,E1 -15979.555,E2 -15979.555} C_VEL
LIN {X 0,Y 475.429,Z 755.184,A -85,B 0,C 180,E1 -15980.005,E2 -15980.005} C_VEL
LIN {X 0,Y 488.36,Z 509.783,A -85,B 0,C 180,E1 -15983.87,E2 -15983.87} C_VEL
LIN {X 0,Y 489.355,Z 489.376,A -85,B 0,C 180,E1 -15984.208,E2 -15984.208} C_VEL
LIN {X 0,Y 478.932,Z 470.966,A -85,B 0,C 180,E1 -15986.445,E2 -15986.445} C_VEL
LIN {X 0,Y 469.028,Z 454.74,A -85,B 0,C 180,E1 -15988.764,E2 -15988.764} C_VEL
LIN {X 0,Y 460.219,Z 441.428,A -85,B 0,C 180,E1 -15991.02,E2 -15991.02} C_VEL
LIN {X 0,Y 452.002,Z 429.482,A -85,B 0,C 180,E1 -15993.352,E2 -15993.352} C_VEL
LIN {X 0,Y 443.501,Z 417.802,A -85,B 0,C 180,E1 -15996.058,E2 -15996.058} C_VEL
LIN {X 0,Y 437.166,Z 409.85,A -85,B 0,C 180,E1 -15998.322,E2 -15998.322} C_VEL
LIN {X 0,Y 433.553,Z 405.907,A -85,B 0,C 180,E1 -15999.725,E2 -15999.725} C_VEL
LIN {X 0,Y 432.144,Z 403.912,A -85,B 0,C 180,E1 -16000.327,E2 -16000.327} C_VEL
LIN {X 0,Y 428.755,Z 400.612,A -85,B 0,C 180,E1 -16001.79,E2 -16001.79} C_VEL
LIN {X 0,Y 427.208,Z 397.957,A -85,B 0,C 180,E1 -16002.567,E2 -16002.567} C_VEL
LIN {X 0,Y 423.776,Z 395.194,A -85,B 0,C 180,E1 -16004.256,E2 -16004.256} C_VEL
LIN {X 0,Y 421.582,Z 391.456,A -85,B 0,C 180,E1 -16005.58,E2 -16005.58} C_VEL
LIN {X 0,Y 418.296,Z 389.37,A -85,B 0,C 180,E1 -16007.576,E2 -16007.576} C_VEL
LIN {X 0,Y 416.219,Z 386.203,A -85,B 0,C 180,E1 -16009.2,E2 -16009.2} C_VEL
LIN {X 0,Y 415.643,Z 384.795,A -85,B 0,C 180,E1 -16009.746,E2 -16009.746} C_VEL
LIN {X 0,Y 411.653,Z 382.447,A -85,B 0,C 180,E1 -16013.725,E2 -16013.725} C_VEL
LIN {X 0,Y 409.599,Z 378.021,A -85,B 0,C 180,E1 -16019.441,E2 -16019.441} C_VEL
LIN {X 0,Y 409.67,Z 378.458,A -85,B 0,C 180,E1 -16021.818,E2 -16021.818} C_VEL
LIN {X 0,Y 413.717,Z 384.101,A -85,B 0,C 180,E1 -16029.038,E2 -16029.038} C_VEL
LIN {X 0,Y 415.845,Z 385.023,A -85,B 0,C 180,E1 -16030.845,E2 -16030.845} C_VEL
LIN {X 0,Y 417.54,Z 388.541,A -85,B 0,C 180,E1 -16032.306,E2 -16032.306} C_VEL
LIN {X 0,Y 420.868,Z 391.185,A -85,B 0,C 180,E1 -16034.445,E2 -16034.445} C_VEL
LIN {X 0,Y 421.794,Z 391.824,A -85,B 0,C 180,E1 -16034.975,E2 -16034.975} C_VEL
LIN {X 0,Y 424.015,Z 395.533,A -85,B 0,C 180,E1 -16036.297,E2 -16036.297} C_VEL
LIN {X 0,Y 427.465,Z 398.398,A -85,B 0,C 180,E1 -16037.985,E2 -16037.985} C_VEL
LIN {X 0,Y 430.321,Z 402.411,A -85,B 0,C 180,E1 -16039.336,E2 -16039.336} C_VEL
LIN {X 0,Y 432.833,Z 404.675,A -85,B 0,C 180,E1 -16040.38,E2 -16040.38} C_VEL
LIN {X 0,Y 435.993,Z 408.875,A -85,B 0,C 180,E1 -16041.668,E2 -16041.668} C_VEL
LIN {X 0,Y 437.998,Z 410.867,A -85,B 0,C 180,E1 -16042.411,E2 -16042.411} C_VEL
LIN {X 0,Y 441.752,Z 415.479,A -85,B 0,C 180,E1 -16043.76,E2 -16043.76} C_VEL
LIN {X 0,Y 447.87,Z 423.045,A -85,B 0,C 180,E1 -16045.772,E2 -16045.772} C_VEL
LIN {X 0,Y 452.929,Z 429.47,A -85,B 0,C 180,E1 -16047.299,E2 -16047.299} C_VEL
LIN {X 0,Y 459.523,Z 437.962,A -85,B 0,C 180,E1 -16049.135,E2 -16049.135} C_VEL
LIN {X 0,Y 469.858,Z 452.111,A -85,B 0,C 180,E1 -16051.747,E2 -16051.747} C_VEL
LIN {X 0,Y 480.921,Z 468.279,A -85,B 0,C 180,E1 -16054.258,E2 -16054.258} C_VEL
LIN {X 0,Y 489.672,Z 482.249,A -85,B 0,C 180,E1 -16056.089,E2 -16056.089} C_VEL
LIN {X 0,Y 476.309,Z 734.526,A -85,B 0,C 180,E1 -16060.048,E2 -16060.048} C_VEL
LIN {X 0,Y 474.479,Z 757.547,A -85,B 0,C 180,E1 -16060.493,E2 -16060.493} C_VEL
LIN {X 0,Y 471.711,Z 781.76,A -85,B 0,C 180,E1 -16061.124,E2 -16061.124} C_VEL
LIN {X 0,Y 468.257,Z 804.179,A -85,B 0,C 180,E1 -16061.906,E2 -16061.906} C_VEL
LIN {X 0,Y 464.318,Z 825.95,A -85,B 0,C 180,E1 -16062.845,E2 -16062.845} C_VEL
LIN {X 0,Y 459.348,Z 849.098,A -85,B 0,C 180,E1 -16064.083,E2 -16064.083} C_VEL
LIN {X 0,Y 454.749,Z 867.962,A -85,B 0,C 180,E1 -16065.283,E2 -16065.283} C_VEL
LIN {X 0,Y 448.669,Z 890.62,A -85,B 0,C 180,E1 -16067.005,E2 -16067.005} C_VEL
LIN {X 0,Y 443.309,Z 908.767,A -85,B 0,C 180,E1 -16068.634,E2 -16068.634} C_VEL
LIN {X 0,Y 437.172,Z 928.36,A -85,B 0,C 180,E1 -16070.688,E2 -16070.688} C_VEL
LIN {X 0,Y 431.5,Z 945.349,A -85,B 0,C 180,E1 -16072.786,E2 -16072.786} C_VEL
LIN {X 0,Y 425.738,Z 962.265,A -85,B 0,C 180,E1 -16075.2,E2 -16075.2} C_VEL
LIN {X 0,Y 420.349,Z 977.646,A -85,B 0,C 180,E1 -16077.803,E2 -16077.803} C_VEL
LIN {X 0,Y 415.443,Z 991.976,A -85,B 0,C 180,E1 -16080.606,E2 -16080.606} C_VEL
LIN {X 0,Y 411.138,Z 1004.676,A -85,B 0,C 180,E1 -16083.573,E2 -16083.573} C_VEL
LIN {X 0,Y 407.507,Z 1016.274,A -85,B 0,C 180,E1 -16086.732,E2 -16086.732} C_VEL
LIN {X 0,Y 404.615,Z 1026.277,A -85,B 0,C 180,E1 -16090.061,E2 -16090.061} C_VEL
LIN {X 0,Y 402.648,Z 1034.317,A -85,B 0,C 180,E1 -16093.258,E2 -16093.258} C_VEL
LIN {X 0,Y 401.232,Z 1041.228,A -85,B 0,C 180,E1 -16096.746,E2 -16096.746} C_VEL
LIN {X 0,Y 400.514,Z 1045.933,A -85,B 0,C 180,E1 -16099.79,E2 -16099.79} C_VEL
LIN {X 0,Y 400.113,Z 1049.913,A -85,B 0,C 180,E1 -16103.399,E2 -16103.399} C_VEL
LIN {X 0,Y 399.992,Z 1051.891,A -85,B 0,C 180,E1 -16106.417,E2 -16106.417} C_VEL
LIN {X 0,Y 399.959,Z 1052.72,A -85,B 0,C 180,E1 -16109.284,E2 -16109.284} C_VEL
LIN {X 0,Y 399.974,Z 1052.338,A -85,B 0,C 180,E1 -16112.723,E2 -16112.723} C_VEL
LIN {X 0,Y 400.062,Z 1050.546,A -85,B 0,C 180,E1 -16115.882,E2 -16115.882} C_VEL
LIN {X 0,Y 400.303,Z 1047.836,A -85,B 0,C 180,E1 -16118.764,E2 -16118.764} C_VEL
LIN {X 0,Y 400.959,Z 1042.895,A -85,B 0,C 180,E1 -16122.384,E2 -16122.384} C_VEL
LIN {X 0,Y 401.148,Z 1041.744,A -85,B 0,C 180,E1 -16123.054,E2 -16123.054} C_VEL
LIN {X 0,Y 400.506,Z 1040.001,A -85,B 0,C 180,E1 -16124.129,E2 -16124.129} C_VEL
LIN {X 0,Y 395.436,Z 1034.682,A -85,B 0,C 180,E1 -16127.09,E2 -16127.09} C_VEL
LIN {X 0,Y 395.256,Z 1032.784,A -85,B 0,C 180,E1 -16127.936,E2 -16127.936} C_VEL
LIN {X 0,Y 397.453,Z 1024.773,A -85,B 0,C 180,E1 -16131.085,E2 -16131.085} C_VEL
LIN {X 0,Y 400.676,Z 1014.29,A -85,B 0,C 180,E1 -16134.472,E2 -16134.472} C_VEL
LIN {X 0,Y 404.076,Z 1004.135,A -85,B 0,C 180,E1 -16137.244,E2 -16137.244} C_VEL
LIN {X 0,Y 408.903,Z 990.53,A -85,B 0,C 180,E1 -16140.41,E2 -16140.41} C_VEL
LIN {X 0,Y 413.599,Z 977.489,A -85,B 0,C 180,E1 -16142.977,E2 -16142.977} C_VEL
LIN {X 0,Y 419.196,Z 962.185,A -85,B 0,C 180,E1 -16145.592,E2 -16145.592} C_VEL
LIN {X 0,Y 425.2,Z 945.206,A -85,B 0,C 180,E1 -16148.033,E2 -16148.033} C_VEL
LIN {X 0,Y 431.095,Z 928.179,A -85,B 0,C 180,E1 -16150.151,E2 -16150.151} C_VEL
LIN {X 0,Y 437.457,Z 908.501,A -85,B 0,C 180,E1 -16152.221,E2 -16152.221} C_VEL
LIN {X 0,Y 443.009,Z 890.3,A -85,B 0,C 180,E1 -16153.861,E2 -16153.861} C_VEL
LIN {X 0,Y 449.132,Z 868.128,A -85,B 0,C 180,E1 -16155.55,E2 -16155.55} C_VEL
LIN {X 0,Y 454.046,Z 848.546,A -85,B 0,C 180,E1 -16156.796,E2 -16156.796} C_VEL
LIN {X 0,Y 459.418,Z 823.838,A -85,B 0,C 180,E1 -16158.102,E2 -16158.102} C_VEL
LIN {X 0,Y 463.304,Z 802.814,A -85,B 0,C 180,E1 -16158.998,E2 -16158.998} C_VEL
LIN {X 0,Y 467.083,Z 777.875,A -85,B 0,C 180,E1 -16159.839,E2 -16159.839} C_VEL
LIN {X 0,Y 469.637,Z 755.562,A -85,B 0,C 180,E1 -16160.401,E2 -16160.401} C_VEL
LIN {X 0,Y 471.639,Z 729.132,A -85,B 0,C 180,E1 -16160.89,E2 -16160.89} C_VEL
LIN {X 0,Y 484.901,Z 486.147,A -85,B 0,C 180,E1 -16164.72,E2 -16164.72} C_VEL
LIN {X 0,Y 474.836,Z 470.429,A -85,B 0,C 180,E1 -16166.912,E2 -16166.912} C_VEL
LIN {X 0,Y 465.569,Z 456.873,A -85,B 0,C 180,E1 -16169.116,E2 -16169.116} C_VEL
LIN {X 0,Y 456.033,Z 443.664,A -85,B 0,C 180,E1 -16171.625,E2 -16171.625} C_VEL
LIN {X 0,Y 448.165,Z 433.432,A -85,B 0,C 180,E1 -16173.926,E2 -16173.926} C_VEL
LIN {X 0,Y 443.68,Z 427.817,A -85,B 0,C 180,E1 -16175.359,E2 -16175.359} C_VEL
LIN {X 0,Y 439.615,Z 422.728,A -85,B 0,C 180,E1 -16176.758,E2 -16176.758} C_VEL
LIN {X 0,Y 435.796,Z 417.812,A -85,B 0,C 180,E1 -16178.18,E2 -16178.18} C_VEL
LIN {X 0,Y 431.915,Z 413.566,A -85,B 0,C 180,E1 -16179.716,E2 -16179.716} C_VEL
LIN {X 0,Y 430.534,Z 411.582,A -85,B 0,C 180,E1 -16180.321,E2 -16180.321} C_VEL
LIN {X 0,Y 426.954,Z 407.877,A -85,B 0,C 180,E1 -16181.922,E2 -16181.922} C_VEL
LIN {X 0,Y 425.562,Z 405.596,A -85,B 0,C 180,E1 -16182.639,E2 -16182.639} C_VEL
LIN {X 0,Y 422.231,Z 402.812,A -85,B 0,C 180,E1 -16184.338,E2 -16184.338} C_VEL
LIN {X 0,Y 420.096,Z 399.233,A -85,B 0,C 180,E1 -16185.668,E2 -16185.668} C_VEL
LIN {X 0,Y 416.568,Z 396.685,A -85,B 0,C 180,E1 -16187.946,E2 -16187.946} C_VEL
LIN {X 0,Y 414.554,Z 392.802,A -85,B 0,C 180,E1 -16189.718,E2 -16189.718} C_VEL
LIN {X 0,Y 410.296,Z 389.984,A -85,B 0,C 180,E1 -16194.406,E2 -16194.406} C_VEL
LIN {X 0,Y 408.844,Z 387.152,A -85,B 0,C 180,E1 -16199.019,E2 -16199.019} C_VEL
LIN {X 0,Y 408.858,Z 387.218,A -85,B 0,C 180,E1 -16200.841,E2 -16200.841} C_VEL
LIN {X 0,Y 409.867,Z 389.436,A -85,B 0,C 180,E1 -16204.477,E2 -16204.477} C_VEL
LIN {X 0,Y 413.959,Z 392.561,A -85,B 0,C 180,E1 -16209.454,E2 -16209.454} C_VEL
LIN {X 0,Y 414.596,Z 392.977,A -85,B 0,C 180,E1 -16210,E2 -16210} C_VEL
LIN {X 0,Y 416.281,Z 396.276,A -85,B 0,C 180,E1 -16211.5,E2 -16211.5} C_VEL
LIN {X 0,Y 419.486,Z 398.975,A -85,B 0,C 180,E1 -16213.649,E2 -16213.649} C_VEL
LIN {X 0,Y 420.373,Z 399.699,A -85,B 0,C 180,E1 -16214.182,E2 -16214.182} C_VEL
LIN {X 0,Y 422.794,Z 403.404,A -85,B 0,C 180,E1 -16215.641,E2 -16215.641} C_VEL
LIN {X 0,Y 425.897,Z 406.152,A -85,B 0,C 180,E1 -16217.206,E2 -16217.206} C_VEL
LIN {X 0,Y 428.839,Z 410.193,A -85,B 0,C 180,E1 -16218.629,E2 -16218.629} C_VEL
LIN {X 0,Y 431.075,Z 412.256,A -85,B 0,C 180,E1 -16219.583,E2 -16219.583} C_VEL
LIN {X 0,Y 434.421,Z 416.564,A -85,B 0,C 180,E1 -16220.972,E2 -16220.972} C_VEL
LIN {X 0,Y 436.215,Z 418.479,A -85,B 0,C 180,E1 -16221.657,E2 -16221.657} C_VEL
LIN {X 0,Y 442.78,Z 426.957,A -85,B 0,C 180,E1 -16224.019,E2 -16224.019} C_VEL
LIN {X 0,Y 451.266,Z 438.891,A -85,B 0,C 180,E1 -16226.731,E2 -16226.731} C_VEL
LIN {X 0,Y 459.151,Z 450.655,A -85,B 0,C 180,E1 -16228.982,E2 -16228.982} C_VEL
LIN {X 0,Y 467.679,Z 464.05,A -85,B 0,C 180,E1 -16231.193,E2 -16231.193} C_VEL
LIN {X 0,Y 476.067,Z 477.972,A -85,B 0,C 180,E1 -16233.189,E2 -16233.189} C_VEL
LIN {X 0,Y 484.68,Z 493.412,A -85,B 0,C 180,E1 -16235.095,E2 -16235.095} C_VEL
LIN {X 0,Y 471.386,Z 738.379,A -85,B 0,C 180,E1 -16238.961,E2 -16238.961} C_VEL
LIN {X 0,Y 469.147,Z 770.305,A -85,B 0,C 180,E1 -16239.527,E2 -16239.527} C_VEL
LIN {X 0,Y 466.598,Z 791.943,A -85,B 0,C 180,E1 -16240.044,E2 -16240.044} C_VEL
LIN {X 0,Y 462.793,Z 816.632,A -85,B 0,C 180,E1 -16240.823,E2 -16240.823} C_VEL
LIN {X 0,Y 458.945,Z 836.983,A -85,B 0,C 180,E1 -16241.644,E2 -16241.644} C_VEL
LIN {X 0,Y 454.359,Z 858.35,A -85,B 0,C 180,E1 -16242.691,E2 -16242.691} C_VEL
LIN {X 0,Y 448.823,Z 880.703,A -85,B 0,C 180,E1 -16244.034,E2 -16244.034} C_VEL
LIN {X 0,Y 443.798,Z 899.071,A -85,B 0,C 180,E1 -16245.336,E2 -16245.336} C_VEL
LIN {X 0,Y 437.202,Z 921.371,A -85,B 0,C 180,E1 -16247.215,E2 -16247.215} C_VEL
LIN {X 0,Y 431.675,Z 938.67,A -85,B 0,C 180,E1 -16248.935,E2 -16248.935} C_VEL
LIN {X 0,Y 425.362,Z 957.653,A -85,B 0,C 180,E1 -16251.124,E2 -16251.124} C_VEL
LIN {X 0,Y 419.381,Z 974.777,A -85,B 0,C 180,E1 -16253.464,E2 -16253.464} C_VEL
LIN {X 0,Y 413.679,Z 991.191,A -85,B 0,C 180,E1 -16256.059,E2 -16256.059} C_VEL
LIN {X 0,Y 408.371,Z 1006.282,A -85,B 0,C 180,E1 -16258.893,E2 -16258.893} C_VEL
LIN {X 0,Y 403.725,Z 1020.205,A -85,B 0,C 180,E1 -16261.929,E2 -16261.929} C_VEL
LIN {X 0,Y 399.945,Z 1032.009,A -85,B 0,C 180,E1 -16265.007,E2 -16265.007} C_VEL
LIN {X 0,Y 397.041,Z 1042.248,A -85,B 0,C 180,E1 -16268.117,E2 -16268.117} C_VEL
LIN {X 0,Y 394.731,Z 1051.556,A -85,B 0,C 180,E1 -16271.54,E2 -16271.54} C_VEL
LIN {X 0,Y 393.333,Z 1058.565,A -85,B 0,C 180,E1 -16274.67,E2 -16274.67} C_VEL
LIN {X 0,Y 392.389,Z 1065.137,A -85,B 0,C 180,E1 -16278.386,E2 -16278.386} C_VEL
LIN {X 0,Y 392.048,Z 1069.175,A -85,B 0,C 180,E1 -16281.493,E2 -16281.493} C_VEL
LIN {X 0,Y 391.953,Z 1072.002,A -85,B 0,C 180,E1 -16284.584,E2 -16284.584} C_VEL
LIN {X 0,Y 391.952,Z 1073.677,A -85,B 0,C 180,E1 -16288.099,E2 -16288.099} C_VEL
LIN {X 0,Y 391.962,Z 1073.816,A -85,B 0,C 180,E1 -16291.023,E2 -16291.023} C_VEL
LIN {X 0,Y 391.946,Z 1072.937,A -85,B 0,C 180,E1 -16293.803,E2 -16293.803} C_VEL
LIN {X 0,Y 391.97,Z 1070.829,A -85,B 0,C 180,E1 -16296.886,E2 -16296.886} C_VEL
LIN {X 0,Y 392.21,Z 1066.811,A -85,B 0,C 180,E1 -16300.428,E2 -16300.428} C_VEL
LIN {X 0,Y 392.77,Z 1062.044,A -85,B 0,C 180,E1 -16303.473,E2 -16303.473} C_VEL
LIN {X 0,Y 393.984,Z 1055.123,A -85,B 0,C 180,E1 -16306.969,E2 -16306.969} C_VEL
LIN {X 0,Y 395.92,Z 1046.452,A -85,B 0,C 180,E1 -16310.396,E2 -16310.396} C_VEL
LIN {X 0,Y 398.671,Z 1036.406,A -85,B 0,C 180,E1 -16313.731,E2 -16313.731} C_VEL
LIN {X 0,Y 402.172,Z 1024.811,A -85,B 0,C 180,E1 -16316.904,E2 -16316.904} C_VEL
LIN {X 0,Y 406.263,Z 1012.451,A -85,B 0,C 180,E1 -16319.812,E2 -16319.812} C_VEL
LIN {X 0,Y 411.434,Z 997.35,A -85,B 0,C 180,E1 -16322.816,E2 -16322.816} C_VEL
LIN {X 0,Y 416.546,Z 982.82,A -85,B 0,C 180,E1 -16325.299,E2 -16325.299} C_VEL
LIN {X 0,Y 422.845,Z 964.703,A -85,B 0,C 180,E1 -16327.938,E2 -16327.938} C_VEL
LIN {X 0,Y 428.489,Z 948.101,A -85,B 0,C 180,E1 -16330.007,E2 -16330.007} C_VEL
LIN {X 0,Y 435.269,Z 927.26,A -85,B 0,C 180,E1 -16332.216,E2 -16332.216} C_VEL
LIN {X 0,Y 440.732,Z 909.372,A -85,B 0,C 180,E1 -16333.826,E2 -16333.826} C_VEL
LIN {X 0,Y 446.798,Z 888.098,A -85,B 0,C 180,E1 -16335.461,E2 -16335.461} C_VEL
LIN {X 0,Y 451.844,Z 868.399,A -85,B 0,C 180,E1 -16336.723,E2 -16336.723} C_VEL
LIN {X 0,Y 456.589,Z 847.854,A -85,B 0,C 180,E1 -16337.841,E2 -16337.841} C_VEL
LIN {X 0,Y 461.405,Z 823.669,A -85,B 0,C 180,E1 -16338.902,E2 -16338.902} C_VEL
LIN {X 0,Y 465.014,Z 802.109,A -85,B 0,C 180,E1 -16339.654,E2 -16339.654} C_VEL
LIN {X 0,Y 468.475,Z 775.771,A -85,B 0,C 180,E1 -16340.346,E2 -16340.346} C_VEL
LIN {X 0,Y 470.41,Z 753.447,A -85,B 0,C 180,E1 -16340.781,E2 -16340.781} C_VEL
LIN {X 0,Y 483.846,Z 506.283,A -85,B 0,C 180,E1 -16344.691,E2 -16344.691} C_VEL
LIN {X 0,Y 484.473,Z 493.176,A -85,B 0,C 180,E1 -16344.915,E2 -16344.915} C_VEL
LIN {X 0,Y 474.828,Z 476.031,A -85,B 0,C 180,E1 -16347.056,E2 -16347.056} C_VEL
LIN {X 0,Y 465.56,Z 460.64,A -85,B 0,C 180,E1 -16349.295,E2 -16349.295} C_VEL
LIN {X 0,Y 457.022,Z 447.539,A -85,B 0,C 180,E1 -16351.549,E2 -16351.549} C_VEL
LIN {X 0,Y 449.254,Z 436.133,A -85,B 0,C 180,E1 -16353.817,E2 -16353.817} C_VEL
LIN {X 0,Y 441.276,Z 424.95,A -85,B 0,C 180,E1 -16356.426,E2 -16356.426} C_VEL
LIN {X 0,Y 435.041,Z 417.124,A -85,B 0,C 180,E1 -16358.706,E2 -16358.706} C_VEL
LIN {X 0,Y 431.443,Z 412.934,A -85,B 0,C 180,E1 -16360.152,E2 -16360.152} C_VEL
LIN {X 0,Y 430.267,Z 411.393,A -85,B 0,C 180,E1 -16360.661,E2 -16360.661} C_VEL
LIN {X 0,Y 426.824,Z 407.778,A -85,B 0,C 180,E1 -16362.199,E2 -16362.199} C_VEL
LIN {X 0,Y 425.419,Z 405.538,A -85,B 0,C 180,E1 -16362.915,E2 -16362.915} C_VEL
LIN {X 0,Y 421.969,Z 402.444,A -85,B 0,C 180,E1 -16364.68,E2 -16364.68} C_VEL
LIN {X 0,Y 419.916,Z 399.166,A -85,B 0,C 180,E1 -16365.943,E2 -16365.943} C_VEL
LIN {X 0,Y 416.752,Z 396.852,A -85,B 0,C 180,E1 -16367.952,E2 -16367.952} C_VEL
LIN {X 0,Y 414.729,Z 393.466,A -85,B 0,C 180,E1 -16369.62,E2 -16369.62} C_VEL
LIN {X 0,Y 414.333,Z 392.664,A -85,B 0,C 180,E1 -16369.994,E2 -16369.994} C_VEL
LIN {X 0,Y 410.115,Z 389.836,A -85,B 0,C 180,E1 -16374.544,E2 -16374.544} C_VEL
LIN {X 0,Y 408.621,Z 386.103,A -85,B 0,C 180,E1 -16379.299,E2 -16379.299} C_VEL
LIN {X 0,Y 408.665,Z 386.225,A -85,B 0,C 180,E1 -16381.542,E2 -16381.542} C_VEL
LIN {X 0,Y 412.608,Z 391.989,A -85,B 0,C 180,E1 -16388.922,E2 -16388.922} C_VEL
LIN {X 0,Y 414.574,Z 392.906,A -85,B 0,C 180,E1 -16390.632,E2 -16390.632} C_VEL
LIN {X 0,Y 416.38,Z 396.465,A -85,B 0,C 180,E1 -16392.2,E2 -16392.2} C_VEL
LIN {X 0,Y 419.686,Z 399.065,A -85,B 0,C 180,E1 -16394.346,E2 -16394.346} C_VEL
LIN {X 0,Y 420.406,Z 399.785,A -85,B 0,C 180,E1 -16394.779,E2 -16394.779} C_VEL
LIN {X 0,Y 422.801,Z 403.491,A -85,B 0,C 180,E1 -16396.204,E2 -16396.204} C_VEL
LIN {X 0,Y 425.879,Z 406.132,A -85,B 0,C 180,E1 -16397.736,E2 -16397.736} C_VEL
LIN {X 0,Y 429.069,Z 410.392,A -85,B 0,C 180,E1 -16399.254,E2 -16399.254} C_VEL
LIN {X 0,Y 431.096,Z 412.321,A -85,B 0,C 180,E1 -16400.112,E2 -16400.112} C_VEL
LIN {X 0,Y 434.55,Z 416.729,A -85,B 0,C 180,E1 -16401.531,E2 -16401.531} C_VEL
LIN {X 0,Y 436.268,Z 418.645,A -85,B 0,C 180,E1 -16402.185,E2 -16402.185} C_VEL
LIN {X 0,Y 441.211,Z 424.763,A -85,B 0,C 180,E1 -16403.968,E2 -16403.968} C_VEL
LIN {X 0,Y 445.946,Z 430.717,A -85,B 0,C 180,E1 -16405.535,E2 -16405.535} C_VEL
LIN {X 0,Y 451.057,Z 437.261,A -85,B 0,C 180,E1 -16407.1,E2 -16407.1} C_VEL
LIN {X 0,Y 457.689,Z 446.059,A -85,B 0,C 180,E1 -16408.976,E2 -16408.976} C_VEL
LIN {X 0,Y 466.942,Z 458.853,A -85,B 0,C 180,E1 -16411.356,E2 -16411.356} C_VEL
LIN {X 0,Y 477.626,Z 474.678,A -85,B 0,C 180,E1 -16413.839,E2 -16413.839} C_VEL
LIN {X 0,Y 484.783,Z 486.274,A -85,B 0,C 180,E1 -16415.384,E2 -16415.384} C_VEL
LIN {X 0,Y 471.117,Z 735.939,A -85,B 0,C 180,E1 -16419.324,E2 -16419.324} C_VEL
LIN {X 0,Y 469.272,Z 758.264,A -85,B 0,C 180,E1 -16419.761,E2 -16419.761} C_VEL
LIN {X 0,Y 466.361,Z 782.742,A -85,B 0,C 180,E1 -16420.407,E2 -16420.407} C_VEL
LIN {X 0,Y 462.902,Z 804.57,A -85,B 0,C 180,E1 -16421.172,E2 -16421.172} C_VEL
LIN {X 0,Y 458.826,Z 826.469,A -85,B 0,C 180,E1 -16422.122,E2 -16422.122} C_VEL
LIN {X 0,Y 453.77,Z 849.32,A -85,B 0,C 180,E1 -16423.351,E2 -16423.351} C_VEL
LIN {X 0,Y 448.807,Z 869.079,A -85,B 0,C 180,E1 -16424.618,E2 -16424.618} C_VEL
LIN {X 0,Y 442.547,Z 891.571,A -85,B 0,C 180,E1 -16426.351,E2 -16426.351} C_VEL
LIN {X 0,Y 437.03,Z 909.651,A -85,B 0,C 180,E1 -16427.994,E2 -16427.994} C_VEL
LIN {X 0,Y 430.398,Z 929.981,A -85,B 0,C 180,E1 -16430.166,E2 -16430.166} C_VEL
LIN {X 0,Y 424.84,Z 946.073,A -85,B 0,C 180,E1 -16432.186,E2 -16432.186} C_VEL
LIN {X 0,Y 418.712,Z 963.323,A -85,B 0,C 180,E1 -16434.697,E2 -16434.697} C_VEL
LIN {X 0,Y 413.421,Z 977.868,A -85,B 0,C 180,E1 -16437.197,E2 -16437.197} C_VEL
LIN {X 0,Y 408.318,Z 992.149,A -85,B 0,C 180,E1 -16440.03,E2 -16440.03} C_VEL
LIN {X 0,Y 403.783,Z 1004.919,A -85,B 0,C 180,E1 -16443.059,E2 -16443.059} C_VEL
LIN {X 0,Y 399.978,Z 1016.495,A -85,B 0,C 180,E1 -16446.267,E2 -16446.267} C_VEL
LIN {X 0,Y 396.926,Z 1026.497,A -85,B 0,C 180,E1 -16449.658,E2 -16449.658} C_VEL
LIN {X 0,Y 394.839,Z 1034.536,A -85,B 0,C 180,E1 -16452.917,E2 -16452.917} C_VEL
LIN {X 0,Y 393.33,Z 1041.446,A -85,B 0,C 180,E1 -16456.475,E2 -16456.475} C_VEL
LIN {X 0,Y 392.557,Z 1046.149,A -85,B 0,C 180,E1 -16459.581,E2 -16459.581} C_VEL
LIN {X 0,Y 392.127,Z 1050.128,A -85,B 0,C 180,E1 -16463.264,E2 -16463.264} C_VEL
LIN {X 0,Y 391.997,Z 1052.105,A -85,B 0,C 180,E1 -16466.344,E2 -16466.344} C_VEL
LIN {X 0,Y 391.962,Z 1052.933,A -85,B 0,C 180,E1 -16469.269,E2 -16469.269} C_VEL
LIN {X 0,Y 391.978,Z 1052.551,A -85,B 0,C 180,E1 -16472.778,E2 -16472.778} C_VEL
LIN {X 0,Y 392.074,Z 1050.76,A -85,B 0,C 180,E1 -16476.002,E2 -16476.002} C_VEL
LIN {X 0,Y 392.328,Z 1048.051,A -85,B 0,C 180,E1 -16478.944,E2 -16478.944} C_VEL
LIN {X 0,Y 393.04,Z 1043.111,A -85,B 0,C 180,E1 -16482.638,E2 -16482.638} C_VEL
LIN {X 0,Y 394.14,Z 1037.496,A -85,B 0,C 180,E1 -16485.751,E2 -16485.751} C_VEL
LIN {X 0,Y 395.256,Z 1032.784,A -85,B 0,C 180,E1 -16487.936,E2 -16487.936} C_VEL
LIN {X 0,Y 394.916,Z 1030.433,A -85,B 0,C 180,E1 -16489.005,E2 -16489.005} C_VEL
LIN {X 0,Y 390.883,Z 1023.86,A -85,B 0,C 180,E1 -16491.896,E2 -16491.896} C_VEL
LIN {X 0,Y 390.958,Z 1021.306,A -85,B 0,C 180,E1 -16492.802,E2 -16492.802} C_VEL
LIN {X 0,Y 394.26,Z 1011.464,A -85,B 0,C 180,E1 -16495.863,E2 -16495.863} C_VEL
LIN {X 0,Y 399.038,Z 998.207,A -85,B 0,C 180,E1 -16499.307,E2 -16499.307} C_VEL
LIN {X 0,Y 403.633,Z 985.902,A -85,B 0,C 180,E1 -16502.014,E2 -16502.014} C_VEL
LIN {X 0,Y 409.685,Z 969.933,A -85,B 0,C 180,E1 -16504.998,E2 -16504.998} C_VEL
LIN {X 0,Y 415.228,Z 955.082,A -85,B 0,C 180,E1 -16507.361,E2 -16507.361} C_VEL
LIN {X 0,Y 421.822,Z 937.007,A -85,B 0,C 180,E1 -16509.824,E2 -16509.824} C_VEL
LIN {X 0,Y 427.688,Z 920.075,A -85,B 0,C 180,E1 -16511.782,E2 -16511.782} C_VEL
LIN {X 0,Y 434.089,Z 900.73,A -85,B 0,C 180,E1 -16513.712,E2 -16513.712} C_VEL
LIN {X 0,Y 439.929,Z 881.166,A -85,B 0,C 180,E1 -16515.349,E2 -16515.349} C_VEL
LIN {X 0,Y 445.124,Z 862.336,A -85,B 0,C 180,E1 -16516.703,E2 -16516.703} C_VEL
LIN {X 0,Y 450.81,Z 839.236,A -85,B 0,C 180,E1 -16518.085,E2 -16518.085} C_VEL
LIN {X 0,Y 455.117,Z 818.925,A -85,B 0,C 180,E1 -16519.093,E2 -16519.093} C_VEL
LIN {X 0,Y 459.589,Z 794.087,A -85,B 0,C 180,E1 -16520.085,E2 -16520.085} C_VEL
LIN {X 0,Y 462.703,Z 772.173,A -85,B 0,C 180,E1 -16520.763,E2 -16520.763} C_VEL
LIN {X 0,Y 465.404,Z 747.205,A -85,B 0,C 180,E1 -16521.342,E2 -16521.342} C_VEL
LIN {X 0,Y 468.964,Z 686.633,A -85,B 0,C 180,E1 -16522.331,E2 -16522.331} C_VEL
LIN {X 0,Y 480.071,Z 490.136,A -85,B 0,C 180,E1 -16525.445,E2 -16525.445} C_VEL
LIN {X 0,Y 470.914,Z 475.779,A -85,B 0,C 180,E1 -16527.507,E2 -16527.507} C_VEL
LIN {X 0,Y 461.6,Z 462.009,A -85,B 0,C 180,E1 -16529.799,E2 -16529.799} C_VEL
LIN {X 0,Y 452.794,Z 449.787,A -85,B 0,C 180,E1 -16532.193,E2 -16532.193} C_VEL
LIN {X 0,Y 445.664,Z 440.363,A -85,B 0,C 180,E1 -16534.341,E2 -16534.341} C_VEL
LIN {X 0,Y 441.259,Z 434.772,A -85,B 0,C 180,E1 -16535.786,E2 -16535.786} C_VEL
LIN {X 0,Y 437.44,Z 429.925,A -85,B 0,C 180,E1 -16537.134,E2 -16537.134} C_VEL
LIN {X 0,Y 433.196,Z 424.624,A -85,B 0,C 180,E1 -16538.753,E2 -16538.753} C_VEL
LIN {X 0,Y 429.545,Z 420.142,A -85,B 0,C 180,E1 -16540.273,E2 -16540.273} C_VEL
LIN {X 0,Y 427.787,Z 418.298,A -85,B 0,C 180,E1 -16541.041,E2 -16541.041} C_VEL
LIN {X 0,Y 424.427,Z 414.018,A -85,B 0,C 180,E1 -16542.661,E2 -16542.661} C_VEL
LIN {X 0,Y 423.526,Z 413.004,A -85,B 0,C 180,E1 -16543.119,E2 -16543.119} C_VEL
LIN {X 0,Y 420.34,Z 409.898,A -85,B 0,C 180,E1 -16544.831,E2 -16544.831} C_VEL
LIN {X 0,Y 418.684,Z 407.013,A -85,B 0,C 180,E1 -16545.901,E2 -16545.901} C_VEL
LIN {X 0,Y 415.236,Z 404.378,A -85,B 0,C 180,E1 -16548.189,E2 -16548.189} C_VEL
LIN {X 0,Y 413.105,Z 400.511,A -85,B 0,C 180,E1 -16550.105,E2 -16550.105} C_VEL
LIN {X 0,Y 409.319,Z 397.972,A -85,B 0,C 180,E1 -16554.393,E2 -16554.393} C_VEL
LIN {X 0,Y 407.869,Z 395.094,A -85,B 0,C 180,E1 -16559.017,E2 -16559.017} C_VEL
LIN {X 0,Y 407.881,Z 395.173,A -85,B 0,C 180,E1 -16560.843,E2 -16560.843} C_VEL
LIN {X 0,Y 408.889,Z 397.432,A -85,B 0,C 180,E1 -16564.488,E2 -16564.488} C_VEL
LIN {X 0,Y 413.158,Z 400.565,A -85,B 0,C 180,E1 -16569.613,E2 -16569.613} C_VEL
LIN {X 0,Y 415.392,Z 404.503,A -85,B 0,C 180,E1 -16571.595,E2 -16571.595} C_VEL
LIN {X 0,Y 418.905,Z 407.382,A -85,B 0,C 180,E1 -16573.915,E2 -16573.915} C_VEL
LIN {X 0,Y 421.463,Z 411.22,A -85,B 0,C 180,E1 -16575.48,E2 -16575.48} C_VEL
LIN {X 0,Y 424.264,Z 413.752,A -85,B 0,C 180,E1 -16576.922,E2 -16576.922} C_VEL
LIN {X 0,Y 427.303,Z 417.882,A -85,B 0,C 180,E1 -16578.415,E2 -16578.415} C_VEL
LIN {X 0,Y 429.354,Z 419.873,A -85,B 0,C 180,E1 -16579.311,E2 -16579.311} C_VEL
LIN {X 0,Y 432.982,Z 424.408,A -85,B 0,C 180,E1 -16580.832,E2 -16580.832} C_VEL
LIN {X 0,Y 434.578,Z 426.34,A -85,B 0,C 180,E1 -16581.459,E2 -16581.459} C_VEL
LIN {X 0,Y 440.382,Z 433.832,A -85,B 0,C 180,E1 -16583.589,E2 -16583.589} C_VEL
LIN {X 0,Y 449.292,Z 446.612,A -85,B 0,C 180,E1 -16586.501,E2 -16586.501} C_VEL
LIN {X 0,Y 457.297,Z 458.869,A -85,B 0,C 180,E1 -16588.825,E2 -16588.825} C_VEL
LIN {X 0,Y 466.155,Z 473.043,A -85,B 0,C 180,E1 -16591.147,E2 -16591.147} C_VEL
LIN {X 0,Y 475.359,Z 488.899,A -85,B 0,C 180,E1 -16593.353,E2 -16593.353} C_VEL
LIN {X 0,Y 479.873,Z 497.388,A -85,B 0,C 180,E1 -16594.378,E2 -16594.378} C_VEL
LIN {X 0,Y 465.832,Z 748.327,A -85,B 0,C 180,E1 -16598.356,E2 -16598.356} C_VEL
LIN {X 0,Y 463.782,Z 772.87,A -85,B 0,C 180,E1 -16598.821,E2 -16598.821} C_VEL
LIN {X 0,Y 460.773,Z 796.918,A -85,B 0,C 180,E1 -16599.418,E2 -16599.418} C_VEL
LIN {X 0,Y 456.865,Z 820.134,A -85,B 0,C 180,E1 -16600.198,E2 -16600.198} C_VEL
LIN {X 0,Y 453.084,Z 839.353,A -85,B 0,C 180,E1 -16600.997,E2 -16600.997} C_VEL
LIN {X 0,Y 447.621,Z 863.388,A -85,B 0,C 180,E1 -16602.226,E2 -16602.226} C_VEL
LIN {X 0,Y 442.61,Z 882.678,A -85,B 0,C 180,E1 -16603.423,E2 -16603.423} C_VEL
LIN {X 0,Y 436.649,Z 903.746,A -85,B 0,C 180,E1 -16604.961,E2 -16604.961} C_VEL
LIN {X 0,Y 430.343,Z 923.844,A -85,B 0,C 180,E1 -16606.731,E2 -16606.731} C_VEL
LIN {X 0,Y 424.45,Z 941.643,A -85,B 0,C 180,E1 -16608.55,E2 -16608.55} C_VEL
LIN {X 0,Y 417.753,Z 960.729,A -85,B 0,C 180,E1 -16610.85,E2 -16610.85} C_VEL
LIN {X 0,Y 412.195,Z 976.145,A -85,B 0,C 180,E1 -16613.016,E2 -16613.016} C_VEL
LIN {X 0,Y 405.65,Z 994.09,A -85,B 0,C 180,E1 -16615.976,E2 -16615.976} C_VEL
LIN {X 0,Y 400.786,Z 1007.48,A -85,B 0,C 180,E1 -16618.572,E2 -16618.572} C_VEL
LIN {X 0,Y 395.593,Z 1022.311,A -85,B 0,C 180,E1 -16621.957,E2 -16621.957} C_VEL
LIN {X 0,Y 392.022,Z 1033.149,A -85,B 0,C 180,E1 -16624.886,E2 -16624.886} C_VEL
LIN {X 0,Y 388.766,Z 1044.204,A -85,B 0,C 180,E1 -16628.42,E2 -16628.42} C_VEL
LIN {X 0,Y 386.671,Z 1052.457,A -85,B 0,C 180,E1 -16631.628,E2 -16631.628} C_VEL
LIN {X 0,Y 385.183,Z 1059.889,A -85,B 0,C 180,E1 -16635.108,E2 -16635.108} C_VEL
LIN {X 0,Y 384.353,Z 1065.554,A -85,B 0,C 180,E1 -16638.597,E2 -16638.597} C_VEL
LIN {X 0,Y 384.035,Z 1069.32,A -85,B 0,C 180,E1 -16641.646,E2 -16641.646} C_VEL
LIN {X 0,Y 383.951,Z 1072.237,A -85,B 0,C 180,E1 -16645.07,E2 -16645.07} C_VEL
LIN {X 0,Y 383.955,Z 1073.51,A -85,B 0,C 180,E1 -16648.358,E2 -16648.358} C_VEL
LIN {X 0,Y 383.962,Z 1073.579,A -85,B 0,C 180,E1 -16651.194,E2 -16651.194} C_VEL
LIN {X 0,Y 383.946,Z 1072.618,A -85,B 0,C 180,E1 -16654.107,E2 -16654.107} C_VEL
LIN {X 0,Y 383.991,Z 1070.09,A -85,B 0,C 180,E1 -16657.631,E2 -16657.631} C_VEL
LIN {X 0,Y 384.283,Z 1066.172,A -85,B 0,C 180,E1 -16660.949,E2 -16660.949} C_VEL
LIN {X 0,Y 384.948,Z 1061.182,A -85,B 0,C 180,E1 -16664.132,E2 -16664.132} C_VEL
LIN {X 0,Y 386.438,Z 1053.465,A -85,B 0,C 180,E1 -16667.933,E2 -16667.933} C_VEL
LIN {X 0,Y 388.412,Z 1045.407,A -85,B 0,C 180,E1 -16671.125,E2 -16671.125} C_VEL
LIN {X 0,Y 391.483,Z 1034.884,A -85,B 0,C 180,E1 -16674.602,E2 -16674.602} C_VEL
LIN {X 0,Y 395.187,Z 1023.425,A -85,B 0,C 180,E1 -16677.746,E2 -16677.746} C_VEL
LIN {X 0,Y 399.799,Z 1010.248,A -85,B 0,C 180,E1 -16680.844,E2 -16680.844} C_VEL
LIN {X 0,Y 404.953,Z 995.867,A -85,B 0,C 180,E1 -16683.684,E2 -16683.684} C_VEL
LIN {X 0,Y 410.874,Z 979.781,A -85,B 0,C 180,E1 -16686.426,E2 -16686.426} C_VEL
LIN {X 0,Y 417.079,Z 962.434,A -85,B 0,C 180,E1 -16688.911,E2 -16688.911} C_VEL
LIN {X 0,Y 423.627,Z 943.945,A -85,B 0,C 180,E1 -16691.187,E2 -16691.187} C_VEL
LIN {X 0,Y 429.884,Z 925.02,A -85,B 0,C 180,E1 -16693.143,E2 -16693.143} C_VEL
LIN {X 0,Y 435.694,Z 906.527,A -85,B 0,C 180,E1 -16694.793,E2 -16694.793} C_VEL
LIN {X 0,Y 441.851,Z 885.162,A -85,B 0,C 180,E1 -16696.398,E2 -16696.398} C_VEL
LIN {X 0,Y 446.827,Z 866.157,A -85,B 0,C 180,E1 -16697.6,E2 -16697.6} C_VEL
LIN {X 0,Y 452.007,Z 844.168,A -85,B 0,C 180,E1 -16698.774,E2 -16698.774} C_VEL
LIN {X 0,Y 456.446,Z 821.833,A -85,B 0,C 180,E1 -16699.727,E2 -16699.727} C_VEL
LIN {X 0,Y 460.314,Z 799.082,A -85,B 0,C 180,E1 -16700.505,E2 -16700.505} C_VEL
LIN {X 0,Y 463.506,Z 774.463,A -85,B 0,C 180,E1 -16701.134,E2 -16701.134} C_VEL
LIN {X 0,Y 465.479,Z 751.71,A -85,B 0,C 180,E1 -16701.574,E2 -16701.574} C_VEL
LIN {X 0,Y 479.393,Z 503.477,A -85,B 0,C 180,E1 -16705.515,E2 -16705.515} C_VEL
LIN {X 0,Y 479.665,Z 496.926,A -85,B 0,C 180,E1 -16705.638,E2 -16705.638} C_VEL
LIN {X 0,Y 470.555,Z 480.675,A -85,B 0,C 180,E1 -16707.731,E2 -16707.731} C_VEL
LIN {X 0,Y 460.847,Z 464.427,A -85,B 0,C 180,E1 -16710.172,E2 -16710.172} C_VEL
LIN {X 0,Y 451.271,Z 449.685,A -85,B 0,C 180,E1 -16712.842,E2 -16712.842} C_VEL
LIN {X 0,Y 445.594,Z 441.476,A -85,B 0,C 180,E1 -16714.586,E2 -16714.586} C_VEL
LIN {X 0,Y 438.896,Z 431.878,A -85,B 0,C 180,E1 -16716.859,E2 -16716.859} C_VEL
LIN {X 0,Y 433.102,Z 424.527,A -85,B 0,C 180,E1 -16719.032,E2 -16719.032} C_VEL
LIN {X 0,Y 429.429,Z 420.074,A -85,B 0,C 180,E1 -16720.551,E2 -16720.551} C_VEL
LIN {X 0,Y 428.105,Z 418.616,A -85,B 0,C 180,E1 -16721.126,E2 -16721.126} C_VEL
LIN {X 0,Y 424.726,Z 414.632,A -85,B 0,C 180,E1 -16722.709,E2 -16722.709} C_VEL
LIN {X 0,Y 423.649,Z 413.089,A -85,B 0,C 180,E1 -16723.265,E2 -16723.265} C_VEL
LIN {X 0,Y 420.187,Z 409.677,A -85,B 0,C 180,E1 -16725.108,E2 -16725.108} C_VEL
LIN {X 0,Y 418.5,Z 406.95,A -85,B 0,C 180,E1 -16726.177,E2 -16726.177} C_VEL
LIN {X 0,Y 415.227,Z 404.324,A -85,B 0,C 180,E1 -16728.33,E2 -16728.33} C_VEL
LIN {X 0,Y 413.334,Z 400.929,A -85,B 0,C 180,E1 -16729.969,E2 -16729.969} C_VEL
LIN {X 0,Y 412.543,Z 400.363,A -85,B 0,C 180,E1 -16730.654,E2 -16730.654} C_VEL
LIN {X 0,Y 408.539,Z 396.893,A -85,B 0,C 180,E1 -16735.649,E2 -16735.649} C_VEL
LIN {X 0,Y 407.637,Z 393.9,A -85,B 0,C 180,E1 -16739.578,E2 -16739.578} C_VEL
LIN {X 0,Y 407.693,Z 394.349,A -85,B 0,C 180,E1 -16741.687,E2 -16741.687} C_VEL
LIN {X 0,Y 411.642,Z 399.951,A -85,B 0,C 180,E1 -16748.943,E2 -16748.943} C_VEL
LIN {X 0,Y 413.347,Z 400.847,A -85,B 0,C 180,E1 -16750.453,E2 -16750.453} C_VEL
LIN {X 0,Y 415.313,Z 404.493,A -85,B 0,C 180,E1 -16752.161,E2 -16752.161} C_VEL
LIN {X 0,Y 418.882,Z 407.372,A -85,B 0,C 180,E1 -16754.48,E2 -16754.48} C_VEL
LIN {X 0,Y 421.467,Z 411.309,A -85,B 0,C 180,E1 -16756.045,E2 -16756.045} C_VEL
LIN {X 0,Y 424.242,Z 413.731,A -85,B 0,C 180,E1 -16757.453,E2 -16757.453} C_VEL
LIN {X 0,Y 427.528,Z 418.082,A -85,B 0,C 180,E1 -16759.042,E2 -16759.042} C_VEL
LIN {X 0,Y 429.371,Z 419.943,A -85,B 0,C 180,E1 -16759.841,E2 -16759.841} C_VEL
LIN {X 0,Y 432.946,Z 424.425,A -85,B 0,C 180,E1 -16761.331,E2 -16761.331} C_VEL
LIN {X 0,Y 434.628,Z 426.51,A -85,B 0,C 180,E1 -16761.988,E2 -16761.988} C_VEL
LIN {X 0,Y 439.18,Z 432.155,A -85,B 0,C 180,E1 -16763.658,E2 -16763.658} C_VEL
LIN {X 0,Y 443.758,Z 437.989,A -85,B 0,C 180,E1 -16765.205,E2 -16765.205} C_VEL
LIN {X 0,Y 450.686,Z 446.896,A -85,B 0,C 180,E1 -16767.339,E2 -16767.339} C_VEL
LIN {X 0,Y 461.089,Z 461.307,A -85,B 0,C 180,E1 -16770.206,E2 -16770.206} C_VEL
LIN {X 0,Y 470.494,Z 475.238,A -85,B 0,C 180,E1 -16772.526,E2 -16772.526} C_VEL
LIN {X 0,Y 479.977,Z 490.11,A -85,B 0,C 180,E1 -16774.661,E2 -16774.661} C_VEL
LIN {X 0,Y 466.064,Z 736.496,A -85,B 0,C 180,E1 -16778.569,E2 -16778.569} C_VEL
LIN {X 0,Y 464.159,Z 758.82,A -85,B 0,C 180,E1 -16779.008,E2 -16779.008} C_VEL
LIN {X 0,Y 461.12,Z 783.509,A -85,B 0,C 180,E1 -16779.666,E2 -16779.666} C_VEL
LIN {X 0,Y 457.623,Z 804.97,A -85,B 0,C 180,E1 -16780.422,E2 -16780.422} C_VEL
LIN {X 0,Y 453.288,Z 827.614,A -85,B 0,C 180,E1 -16781.411,E2 -16781.411} C_VEL
LIN {X 0,Y 448.114,Z 850.171,A -85,B 0,C 180,E1 -16782.639,E2 -16782.639} C_VEL
LIN {X 0,Y 442.929,Z 870.196,A -85,B 0,C 180,E1 -16783.935,E2 -16783.935} C_VEL
LIN {X 0,Y 436.732,Z 891.72,A -85,B 0,C 180,E1 -16785.609,E2 -16785.609} C_VEL
LIN {X 0,Y 431.052,Z 909.758,A -85,B 0,C 180,E1 -16787.258,E2 -16787.258} C_VEL
LIN {X 0,Y 424.073,Z 930.455,A -85,B 0,C 180,E1 -16789.49,E2 -16789.49} C_VEL
LIN {X 0,Y 418.227,Z 946.797,A -85,B 0,C 180,E1 -16791.567,E2 -16791.567} C_VEL
LIN {X 0,Y 411.589,Z 964.721,A -85,B 0,C 180,E1 -16794.233,E2 -16794.233} C_VEL
LIN {X 0,Y 406.255,Z 978.852,A -85,B 0,C 180,E1 -16796.712,E2 -16796.712} C_VEL
LIN {X 0,Y 400.723,Z 993.633,A -85,B 0,C 180,E1 -16799.733,E2 -16799.733} C_VEL
LIN {X 0,Y 396.275,Z 1005.685,A -85,B 0,C 180,E1 -16802.663,E2 -16802.663} C_VEL
LIN {X 0,Y 392.315,Z 1017.187,A -85,B 0,C 180,E1 -16805.934,E2 -16805.934} C_VEL
LIN {X 0,Y 389.258,Z 1026.717,A -85,B 0,C 180,E1 -16809.238,E2 -16809.238} C_VEL
LIN {X 0,Y 386.961,Z 1035.102,A -85,B 0,C 180,E1 -16812.713,E2 -16812.713} C_VEL
LIN {X 0,Y 385.434,Z 1041.663,A -85,B 0,C 180,E1 -16816.192,E2 -16816.192} C_VEL
LIN {X 0,Y 384.603,Z 1046.366,A -85,B 0,C 180,E1 -16819.363,E2 -16819.363} C_VEL
LIN {X 0,Y 384.142,Z 1050.343,A -85,B 0,C 180,E1 -16823.123,E2 -16823.123} C_VEL
LIN {X 0,Y 384.003,Z 1052.319,A -85,B 0,C 180,E1 -16826.268,E2 -16826.268} C_VEL
LIN {X 0,Y 383.965,Z 1053.147,A -85,B 0,C 180,E1 -16829.254,E2 -16829.254} C_VEL
LIN {X 0,Y 383.982,Z 1052.765,A -85,B 0,C 180,E1 -16832.836,E2 -16832.836} C_VEL
LIN {X 0,Y 384.089,Z 1050.974,A -85,B 0,C 180,E1 -16836.127,E2 -16836.127} C_VEL
LIN {X 0,Y 384.353,Z 1048.266,A -85,B 0,C 180,E1 -16839.131,E2 -16839.131} C_VEL
LIN {X 0,Y 385.084,Z 1043.576,A -85,B 0,C 180,E1 -16842.751,E2 -16842.751} C_VEL
LIN {X 0,Y 386.299,Z 1037.713,A -85,B 0,C 180,E1 -16846.079,E2 -16846.079} C_VEL
LIN {X 0,Y 388.309,Z 1030.132,A -85,B 0,C 180,E1 -16849.557,E2 -16849.557} C_VEL
LIN {X 0,Y 390.958,Z 1021.306,A -85,B 0,C 180,E1 -16852.802,E2 -16852.802} C_VEL
LIN {X 0,Y 391.01,Z 1018.357,A -85,B 0,C 180,E1 -16853.853,E2 -16853.853} C_VEL
LIN {X 0,Y 388.07,Z 1010.414,A -85,B 0,C 180,E1 -16856.721,E2 -16856.721} C_VEL
LIN {X 0,Y 388.467,Z 1007.407,A -85,B 0,C 180,E1 -16857.598,E2 -16857.598} C_VEL
LIN {X 0,Y 392.767,Z 996.135,A -85,B 0,C 180,E1 -16860.438,E2 -16860.438} C_VEL
LIN {X 0,Y 398.404,Z 981.844,A -85,B 0,C 180,E1 -16863.514,E2 -16863.514} C_VEL
LIN {X 0,Y 403.947,Z 967.64,A -85,B 0,C 180,E1 -16866.095,E2 -16866.095} C_VEL
LIN {X 0,Y 410.394,Z 951.156,A -85,B 0,C 180,E1 -16868.678,E2 -16868.678} C_VEL
LIN {X 0,Y 416.912,Z 933.562,A -85,B 0,C 180,E1 -16870.991,E2 -16870.991} C_VEL
LIN {X 0,Y 423.383,Z 915.458,A -85,B 0,C 180,E1 -16873.041,E2 -16873.041} C_VEL
LIN {X 0,Y 429.834,Z 895.834,A -85,B 0,C 180,E1 -16874.911,E2 -16874.911} C_VEL
LIN {X 0,Y 435.473,Z 877.342,A -85,B 0,C 180,E1 -16876.421,E2 -16876.421} C_VEL
LIN {X 0,Y 441.795,Z 854.356,A -85,B 0,C 180,E1 -16877.99,E2 -16877.99} C_VEL
LIN {X 0,Y 446.499,Z 834.942,A -85,B 0,C 180,E1 -16879.095,E2 -16879.095} C_VEL
LIN {X 0,Y 451.278,Z 812.473,A -85,B 0,C 180,E1 -16880.161,E2 -16880.161} C_VEL
LIN {X 0,Y 455.128,Z 790.218,A -85,B 0,C 180,E1 -16880.996,E2 -16880.996} C_VEL
LIN {X 0,Y 458.28,Z 768.003,A -85,B 0,C 180,E1 -16881.656,E2 -16881.656} C_VEL
LIN {X 0,Y 460.776,Z 742.905,A -85,B 0,C 180,E1 -16882.2,E2 -16882.2} C_VEL
LIN {X 0,Y 474.488,Z 508.922,A -85,B 0,C 180,E1 -16885.94,E2 -16885.94} C_VEL
LIN {X 0,Y 475.269,Z 494.043,A -85,B 0,C 180,E1 -16886.195,E2 -16886.195} C_VEL
LIN {X 0,Y 465.36,Z 478.486,A -85,B 0,C 180,E1 -16888.525,E2 -16888.525} C_VEL
LIN {X 0,Y 454.889,Z 463.089,A -85,B 0,C 180,E1 -16891.26,E2 -16891.26} C_VEL
